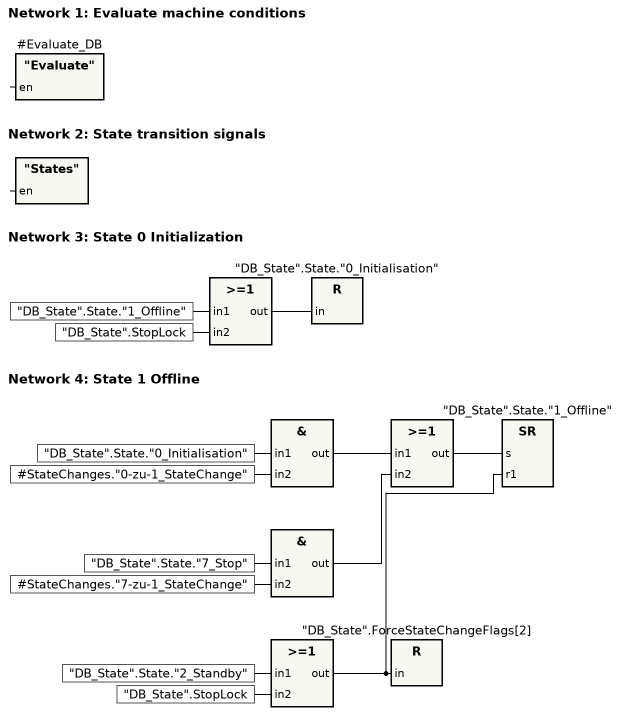
   #Evaluate_DB();   // "Evaluate"
END_REGION

REGION Network 2: State transition signals
   "States"();
END_REGION

REGION Network 3: State 0 Initialization
   // The "missing" SET logic is here:
   // Initialise (FB25) NW 2: "DB_StateMachine".State."0_Initialisation" := TRUE;
   IF "DB_State".State."1_Offline" OR "DB_State".StopLock THEN
       "DB_State".State."0_Initialisation" := FALSE;
   END_IF;
END_REGION

REGION Network 4: State 1 Offline
   #_w1 := "DB_State".State."2_Standby" OR "DB_State".StopLock;
   IF ("DB_State".State."0_Initialisation" AND #StateChanges."0-zu-1_StateChange") OR ("DB_State".State."7_Stop" AND #StateChanges."7-zu-1_StateChange") THEN
       "DB_State".State."1_Offline" := TRUE;   // SR flip-flop
   END_IF;
   IF #_w1 THEN
       "DB_State".State."1_Offline" := FALSE;
       "DB_State".ForceStateChangeFlags[2] := FALSE;
   END_IF;
END_REGION

REGION Network 5: State 2 Standby
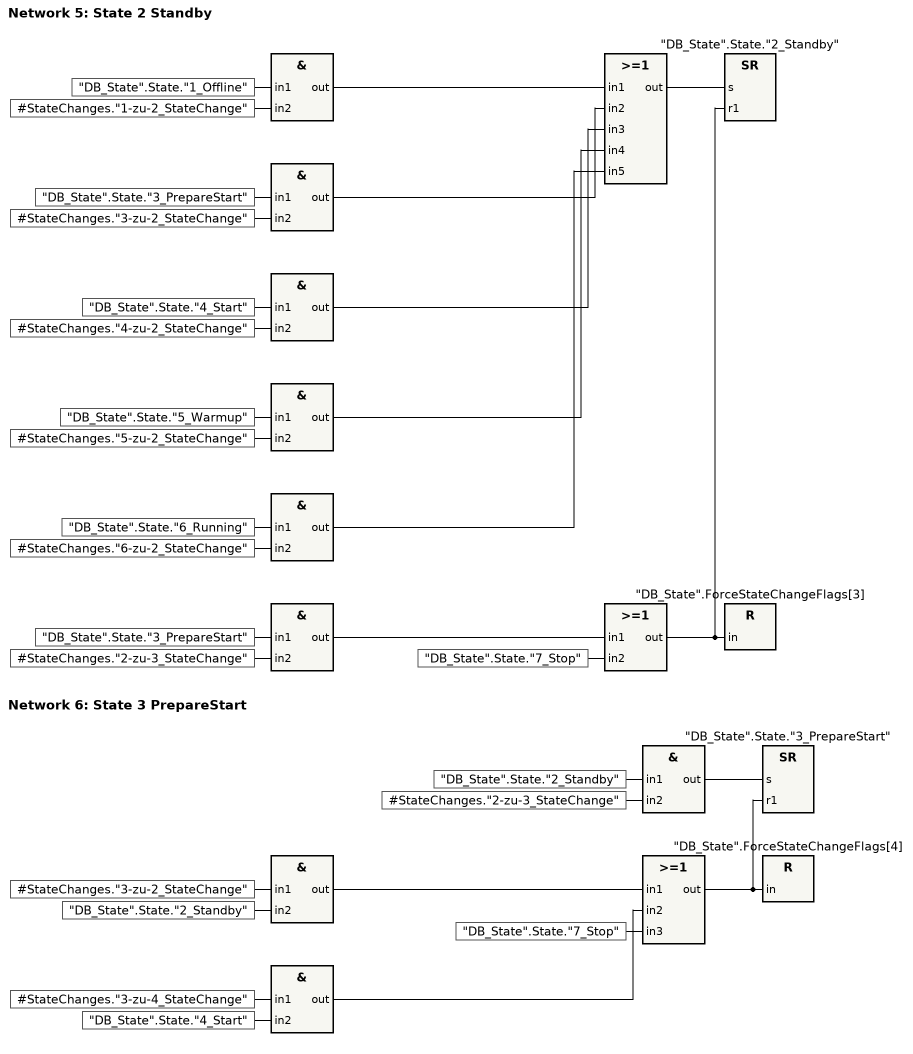
   #_w1 := ("DB_State".State."3_PrepareStart" AND #StateChanges."2-zu-3_StateChange") OR "DB_State".State."7_Stop";
   IF ("DB_State".State."1_Offline" AND #StateChanges."1-zu-2_StateChange") OR ("DB_State".State."3_PrepareStart" AND #StateChanges."3-zu-2_StateChange") OR ("DB_State".State."4_Start" AND #StateChanges."4-zu-2_StateChange") OR ("DB_State".State."5_Warmup" AND #StateChanges."5-zu-2_StateChange") OR ("DB_State".State."6_Running" AND #StateChanges."6-zu-2_StateChange") THEN
       "DB_State".State."2_Standby" := TRUE;   // SR flip-flop
   END_IF;
   IF #_w1 THEN
       "DB_State".State."2_Standby" := FALSE;
       "DB_State".ForceStateChangeFlags[3] := FALSE;
   END_IF;
END_REGION

REGION Network 6: State 3 PrepareStart
   #_w1 := (#StateChanges."3-zu-2_StateChange" AND "DB_State".State."2_Standby") OR (#StateChanges."3-zu-4_StateChange" AND "DB_State".State."4_Start") OR "DB_State".State."7_Stop";
   IF "DB_State".State."2_Standby" AND #StateChanges."2-zu-3_StateChange" THEN
       "DB_State".State."3_PrepareStart" := TRUE;   // SR flip-flop
   END_IF;
   IF #_w1 THEN
       "DB_State".State."3_PrepareStart" := FALSE;
       "DB_State".ForceStateChangeFlags[4] := FALSE;
   END_IF;
END_REGION

REGION Network 7: State 4 Start
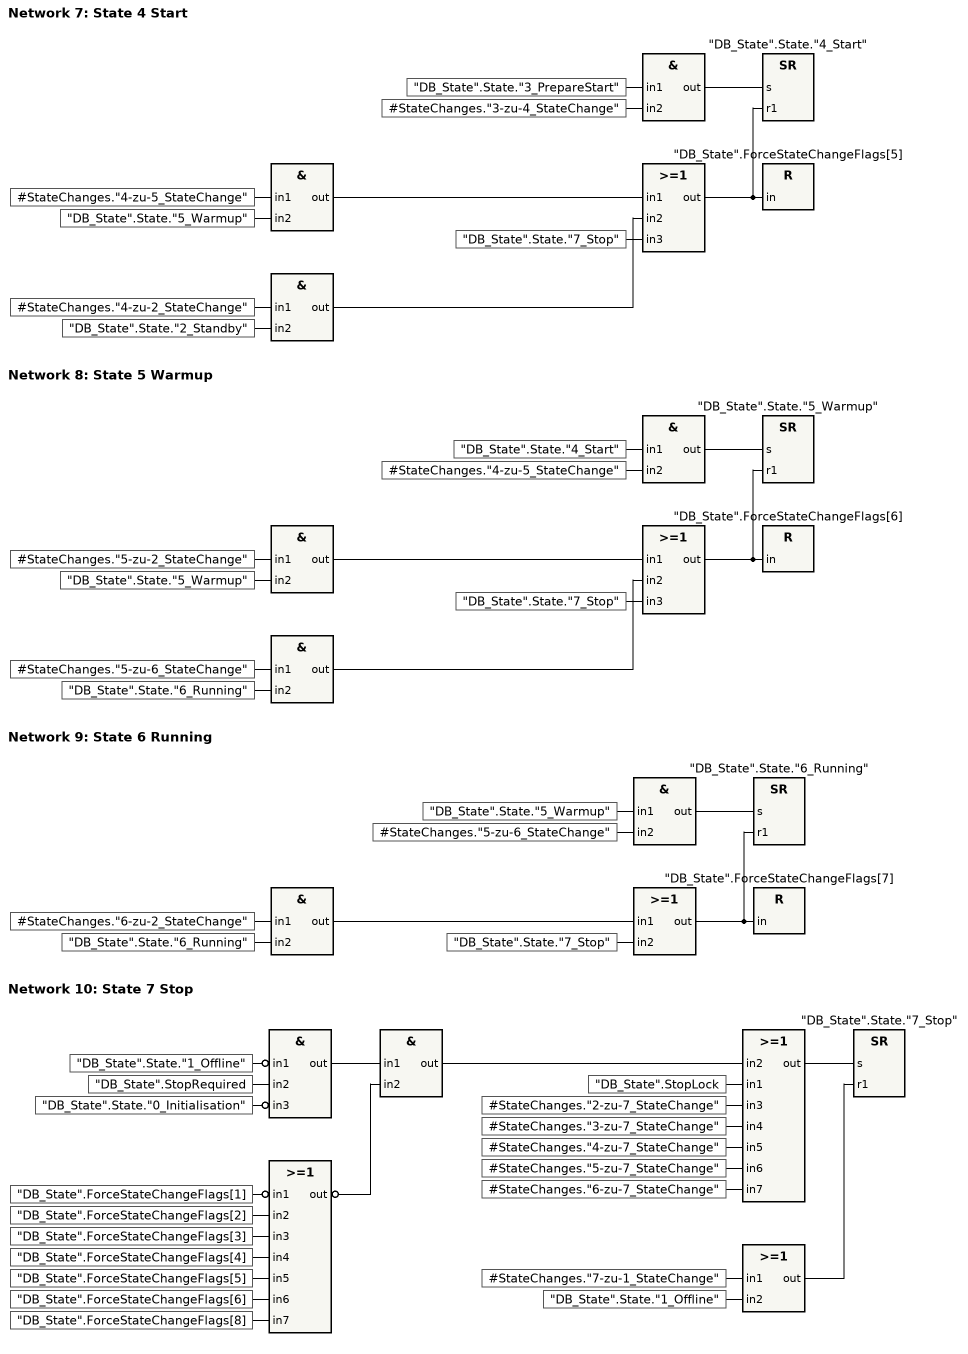
   #_w1 := (#StateChanges."4-zu-5_StateChange" AND "DB_State".State."5_Warmup") OR (#StateChanges."4-zu-2_StateChange" AND "DB_State".State."2_Standby") OR "DB_State".State."7_Stop";
   IF "DB_State".State."3_PrepareStart" AND #StateChanges."3-zu-4_StateChange" THEN
       "DB_State".State."4_Start" := TRUE;   // SR flip-flop
   END_IF;
   IF #_w1 THEN
       "DB_State".State."4_Start" := FALSE;
       "DB_State".ForceStateChangeFlags[5] := FALSE;
   END_IF;
END_REGION

REGION Network 8: State 5 Warmup
   #_w1 := (#StateChanges."5-zu-2_StateChange" AND "DB_State".State."5_Warmup") OR (#StateChanges."5-zu-6_StateChange" AND "DB_State".State."6_Running") OR "DB_State".State."7_Stop";
   IF "DB_State".State."4_Start" AND #StateChanges."4-zu-5_StateChange" THEN
       "DB_State".State."5_Warmup" := TRUE;   // SR flip-flop
   END_IF;
   IF #_w1 THEN
       "DB_State".State."5_Warmup" := FALSE;
       "DB_State".ForceStateChangeFlags[6] := FALSE;
   END_IF;
END_REGION

REGION Network 9: State 6 Running
   #_w1 := (#StateChanges."6-zu-2_StateChange" AND "DB_State".State."6_Running") OR "DB_State".State."7_Stop";
   IF "DB_State".State."5_Warmup" AND #StateChanges."5-zu-6_StateChange" THEN
       "DB_State".State."6_Running" := TRUE;   // SR flip-flop
   END_IF;
   IF #_w1 THEN
       "DB_State".State."6_Running" := FALSE;
       "DB_State".ForceStateChangeFlags[7] := FALSE;
   END_IF;
END_REGION

REGION Network 10: State 7 Stop
   IF (NOT "DB_State".State."1_Offline" AND "DB_State".StopRequired AND NOT "DB_State".State."0_Initialisation" AND NOT (NOT "DB_State".ForceStateChangeFlags[1] OR "DB_State".ForceStateChangeFlags[2] OR "DB_State".ForceStateChangeFlags[3] OR "DB_State".ForceStateChangeFlags[4] OR "DB_State".ForceStateChangeFlags[5] OR "DB_State".ForceStateChangeFlags[6] OR "DB_State".ForceStateChangeFlags[8])) OR "DB_State".StopLock OR #StateChanges."2-zu-7_StateChange" OR #StateChanges."3-zu-7_StateChange" OR #StateChanges."4-zu-7_StateChange" OR #StateChanges."5-zu-7_StateChange" OR #StateChanges."6-zu-7_StateChange" THEN
       "DB_State".State."7_Stop" := TRUE;   // SR flip-flop
   END_IF;
   IF #StateChanges."7-zu-1_StateChange" OR "DB_State".State."1_Offline" THEN
       "DB_State".State."7_Stop" := FALSE;
   END_IF;
END_REGION
END_FUNCTION_BLOCK

FUNCTION_BLOCK "Evaluate"   // FB26, FBD
TITLE = Evaluate machine state conditions
{ S7_Optimized_Access := 'TRUE' }
AUTHOR : Heaten
VERSION : 0.1
// stored: AutoNumber true, IsIECCheckEnabled false, IsRetainMemResEnabled false, MemoryReserve 0, SetENOAutomatically false, UDAEnableTagReadback false
   VAR
      TOF2_StandbyPauseTime { S7_SetPoint := 'True'} : TOF_TIME;
      TON2_Standby { S7_SetPoint := 'True'} : TON_TIME;
      TON3_PrepareStart { S7_SetPoint := 'True'} : TON_TIME;
      TON4_Start { S7_SetPoint := 'True'} : TON_TIME;
      TON5_Warmup { S7_SetPoint := 'True'} : TON_TIME;
      TON7_Stop { S7_SetPoint := 'True'} : TON_TIME;
      MinimumPriming { S7_SetPoint := 'True'} : TON_TIME;
   END_VAR
   VAR_TEMP
      HydrolockSpeed : Real;
      HeatSinkTemperatureMax : Real;
   END_VAR
BEGIN

REGION Network 1: Check running condition: system initialized
   // Add more conditions here
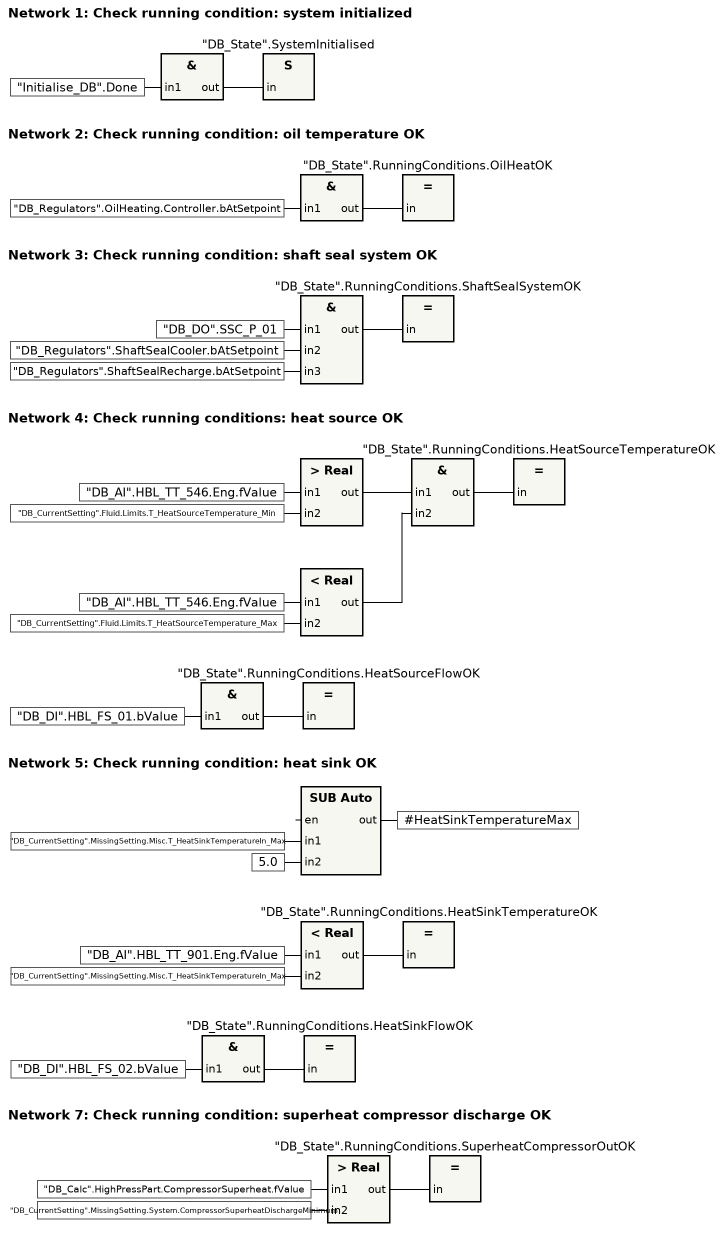
   IF "Initialise_DB".Done THEN "DB_State".SystemInitialised := TRUE; END_IF;
END_REGION

REGION Network 2: Check running condition: oil temperature OK
   "DB_State".RunningConditions.OilHeatOK := "DB_Regulators".OilHeating.Controller.bAtSetpoint;
END_REGION

REGION Network 3: Check running condition: shaft seal system OK
   "DB_State".RunningConditions.ShaftSealSystemOK := "DB_DO".SSC_P_01 AND "DB_Regulators".ShaftSealCooler.bAtSetpoint AND "DB_Regulators".ShaftSealRecharge.bAtSetpoint;
END_REGION

REGION Network 4: Check running conditions: heat source OK
   "DB_State".RunningConditions.HeatSourceTemperatureOK := ("DB_AI".HBL_TT_546.Eng.fValue > "DB_CurrentSetting".Fluid.Limits.T_HeatSourceTemperature_Min) AND ("DB_AI".HBL_TT_546.Eng.fValue < "DB_CurrentSetting".Fluid.Limits.T_HeatSourceTemperature_Max);
   "DB_State".RunningConditions.HeatSourceFlowOK := "DB_DI".HBL_FS_01.bValue;
END_REGION

REGION Network 5: Check running condition: heat sink OK
   // NOTE: leave a little headroom to the limit for standby, otherwise the machine shuts down (via alarm 2101) at the same temperature as it should go to standby on
   #HeatSinkTemperatureMax := "DB_CurrentSetting".MissingSetting.Misc.T_HeatSinkTemperatureIn_Max - 5.0;
   "DB_State".RunningConditions.HeatSinkTemperatureOK := "DB_AI".HBL_TT_901.Eng.fValue < "DB_CurrentSetting".MissingSetting.Misc.T_HeatSinkTemperatureIn_Max;
   "DB_State".RunningConditions.HeatSinkFlowOK := "DB_DI".HBL_FS_02.bValue;
END_REGION

REGION Network 6 (SCL): Check running condition: recuperator working
   // Recuperator sits between evaporator and compressor and SHOULD INCREASE THE SUPERHEAT (ie delta T over the recuperator should be positive)
   // 
   // Recuperator window: must add at least "DB_CurrentSetting".MissingSetting.System.RecuperatorSuperheatGainWorking degrees to be considered working, 
   // but can then fall as low as "DB_CurrentSetting".MissingSetting.System.RecuperatorSuperheatGainNotWorking degrees before it is considered not working again
   (*
   IF ("DB_Calc".LowPressPart.CompressorSuperheat.fValue - 2) <      //If the superheat at compressor inlet minus 2 is smaller than
       "DB_Calc".LowPressPart.EvaporatorSuperheat.fValue THEN          //the superheat at the evaporator, the recuperator doesn´t work
       "StateMachine_DB".RunningConditions.RecuperatorWorking := FALSE;
   ELSIF
       ("DB_Calc".LowPressPart.CompressorSuperheat.fValue + 3) >     //If the superheat at compressor inlet plus 3 is bigger than
       "DB_Calc".LowPressPart.EvaporatorSuperheat.fValue THEN          //the superheat at the evaporator, the recuperator works
       "StateMachine_DB".RunningConditions.RecuperatorWorking := TRUE;
   END_IF;
   *)

   // Rewritten with user-defined limits and right-side-up logic
   // Also don't evaluate the condition unless it's relevant, to avoid odd conditions during earlier states/cold start setting this accidentally
   IF "DB_State".State.State_Number = 5 OR "DB_State".State.State_Number = 6 THEN
       IF "DB_Calc".LowPressPart.CompressorSuperheat.fValue > "DB_Calc".LowPressPart.EvaporatorSuperheat.fValue + "DB_CurrentSetting".MissingSetting.System.RecuperatorDeltaTWorking THEN
           "DB_State".RunningConditions.RecuperatorWorking := TRUE;
       ELSIF "DB_Calc".LowPressPart.CompressorSuperheat.fValue < "DB_Calc".LowPressPart.EvaporatorSuperheat.fValue + "DB_CurrentSetting".MissingSetting.System.RecuperatorDeltaTNotWorking THEN
           "DB_State".RunningConditions.RecuperatorWorking := FALSE;
       END_IF;
   ELSE
       "DB_State".RunningConditions.RecuperatorWorking := FALSE;
   END_IF;
END_REGION

REGION Network 7: Check running condition: superheat compressor discharge OK
   "DB_State".RunningConditions.SuperheatCompressorOutOK := "DB_Calc".HighPressPart.CompressorSuperheat.fValue > "DB_CurrentSetting".MissingSetting.System.CompressorSuperheatDischargeMinimum;
END_REGION

REGION Network 8: Check running condition: at or above hydrolock speed
   // Give a small margin for error, so if it sits at, for example 288.2 RPM and the limit is 290, it will work.
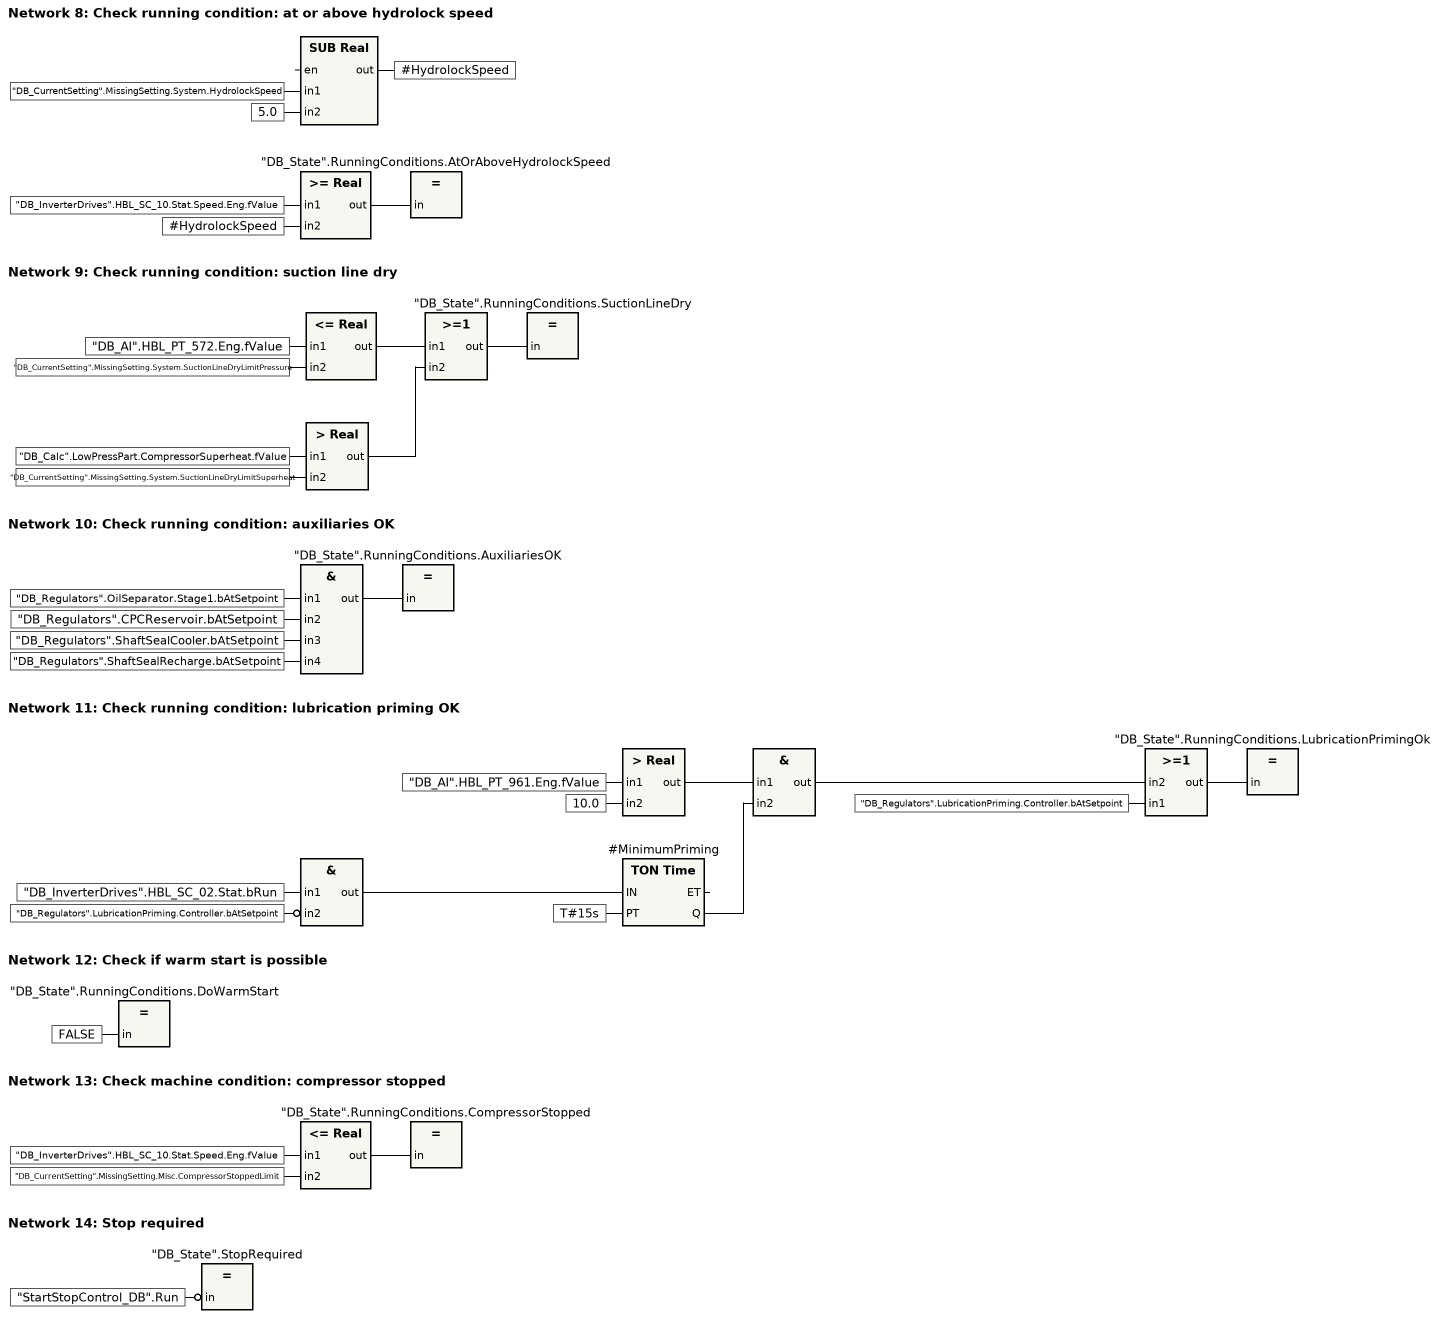
   #HydrolockSpeed := "DB_CurrentSetting".MissingSetting.System.HydrolockSpeed - 5.0;
   "DB_State".RunningConditions.AtOrAboveHydrolockSpeed := "DB_InverterDrives".HBL_SC_10.Stat.Speed.Eng.fValue >= #HydrolockSpeed;
END_REGION

REGION Network 9: Check running condition: suction line dry
   "DB_State".RunningConditions.SuctionLineDry := ("DB_AI".HBL_PT_572.Eng.fValue <= "DB_CurrentSetting".MissingSetting.System.SuctionLineDryLimitPressure) OR ("DB_Calc".LowPressPart.CompressorSuperheat.fValue > "DB_CurrentSetting".MissingSetting.System.SuctionLineDryLimitSuperheat);
END_REGION

REGION Network 10: Check running condition: auxiliaries OK
   "DB_State".RunningConditions.AuxiliariesOK := "DB_Regulators".OilSeparator.Stage1.bAtSetpoint AND "DB_Regulators".CPCReservoir.bAtSetpoint AND "DB_Regulators".ShaftSealCooler.bAtSetpoint AND "DB_Regulators".ShaftSealRecharge.bAtSetpoint;
END_REGION

REGION Network 11: Check running condition: lubrication priming OK
   // The simplest is to just look at the regulator's .bAtSetpoint bit. But the lubrication priming pump may be too small to reach the setpoint. So a hybrid condition is:
   // IF the pressure is at setpoint OR
   // the motor has been running for at least X sec when not at setpoint AND 
   // the developed lubrication pressure is greater than Y kPa THEN
   // the lubrication system is working ok.
   // NOTE: hardcoded params = bad!!
   #MinimumPriming(IN := "DB_InverterDrives".HBL_SC_02.Stat.bRun AND NOT "DB_Regulators".LubricationPriming.Controller.bAtSetpoint,   // TON
                   PT := T#15s);
   "DB_State".RunningConditions.LubricationPrimingOk := (("DB_AI".HBL_PT_961.Eng.fValue > 10.0) AND #MinimumPriming.Q) OR "DB_Regulators".LubricationPriming.Controller.bAtSetpoint;
END_REGION

REGION Network 12: Check if warm start is possible
   // Think of an appropriate condition
   "DB_State".RunningConditions.DoWarmStart := FALSE;
END_REGION

REGION Network 13: Check machine condition: compressor stopped
   "DB_State".RunningConditions.CompressorStopped := "DB_InverterDrives".HBL_SC_10.Stat.Speed.Eng.fValue <= "DB_CurrentSetting".MissingSetting.Misc.CompressorStoppedLimit;
END_REGION

REGION Network 14: Stop required
   // NOte: stop conditions are evaluated by FB30 StartStopControl
   "DB_State".StopRequired := NOT "StartStopControl_DB".Run;
END_REGION

REGION Network 15: Check for risk of hydrolock
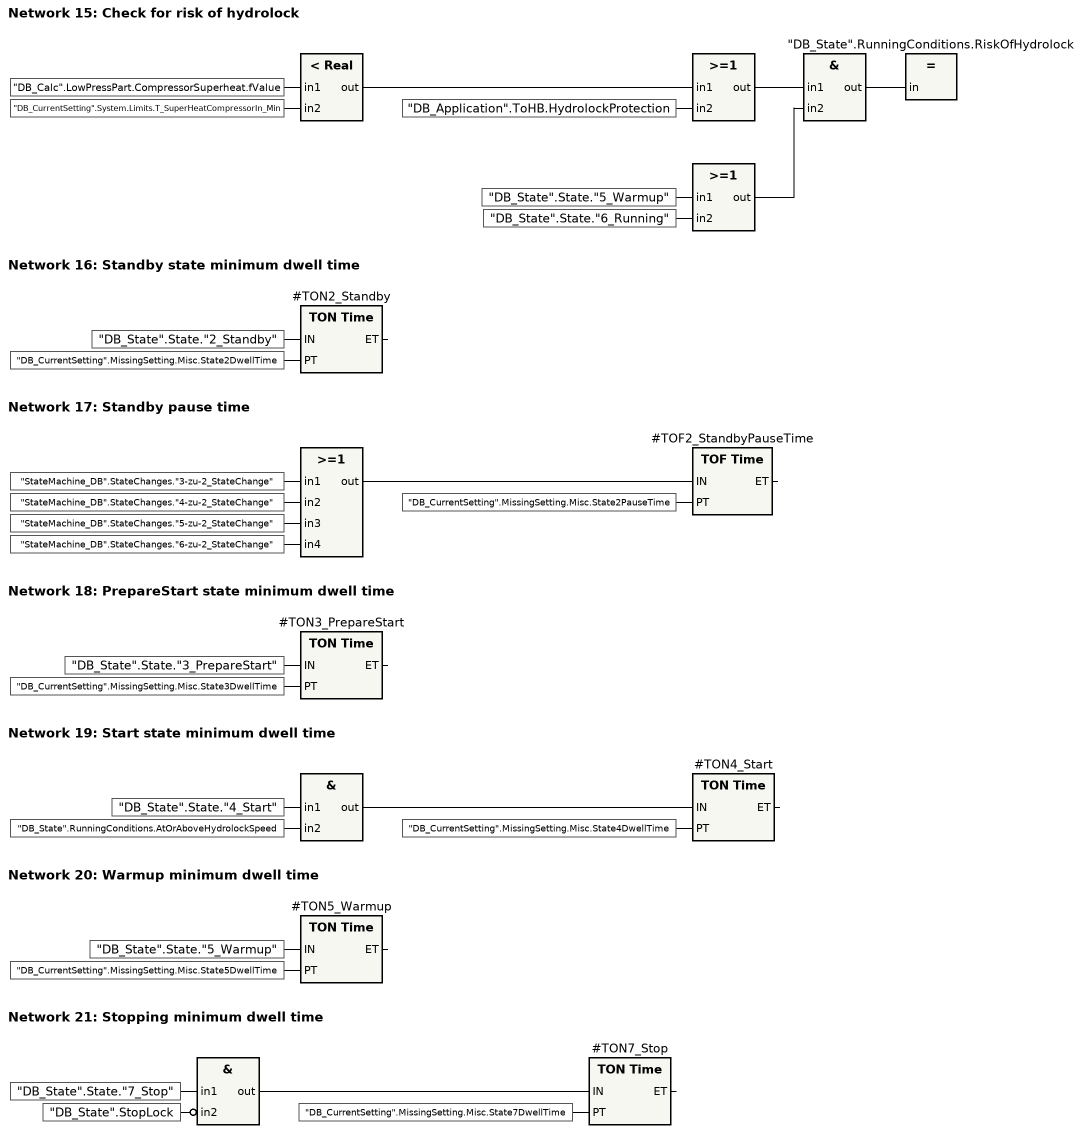
   "DB_State".RunningConditions.RiskOfHydrolock := (("DB_Calc".LowPressPart.CompressorSuperheat.fValue < "DB_CurrentSetting".System.Limits.T_SuperHeatCompressorIn_Min) OR "DB_Application".ToHB.HydrolockProtection) AND ("DB_State".State."5_Warmup" OR "DB_State".State."6_Running");
END_REGION

REGION Network 16: Standby state minimum dwell time
   #TON2_Standby(IN := "DB_State".State."2_Standby",   // TON
                 PT := "DB_CurrentSetting".MissingSetting.Misc.State2DwellTime);
END_REGION

REGION Network 17: Standby pause time
   // Minimum pause in Standby before resume
   #TOF2_StandbyPauseTime(IN := "StateMachine_DB".StateChanges."3-zu-2_StateChange" OR "StateMachine_DB".StateChanges."4-zu-2_StateChange" OR "StateMachine_DB".StateChanges."5-zu-2_StateChange" OR "StateMachine_DB".StateChanges."6-zu-2_StateChange",   // TOF
                          PT := "DB_CurrentSetting".MissingSetting.Misc.State2PauseTime);
END_REGION

REGION Network 18: PrepareStart state minimum dwell time
   #TON3_PrepareStart(IN := "DB_State".State."3_PrepareStart",   // TON
                      PT := "DB_CurrentSetting".MissingSetting.Misc.State3DwellTime);
END_REGION

REGION Network 19: Start state minimum dwell time
   #TON4_Start(IN := "DB_State".State."4_Start" AND "DB_State".RunningConditions.AtOrAboveHydrolockSpeed,   // TON
               PT := "DB_CurrentSetting".MissingSetting.Misc.State4DwellTime);
END_REGION

REGION Network 20: Warmup minimum dwell time
   #TON5_Warmup(IN := "DB_State".State."5_Warmup",   // TON
                PT := "DB_CurrentSetting".MissingSetting.Misc.State5DwellTime);
END_REGION

REGION Network 21: Stopping minimum dwell time
   #TON7_Stop(IN := "DB_State".State."7_Stop" AND NOT "DB_State".StopLock,   // TON
              PT := "DB_CurrentSetting".MissingSetting.Misc.State7DwellTime);
END_REGION
END_FUNCTION_BLOCK

FUNCTION "States" : Void   // FC27, FBD
TITLE = State change signal generation
{ S7_Optimized_Access := 'TRUE' }
VERSION : 0.1
// stored: AutoNumber true, IsIECCheckEnabled false, SetENOAutomatically false, UDAEnableTagReadback false
BEGIN

REGION Network 1: State 0 Initialization
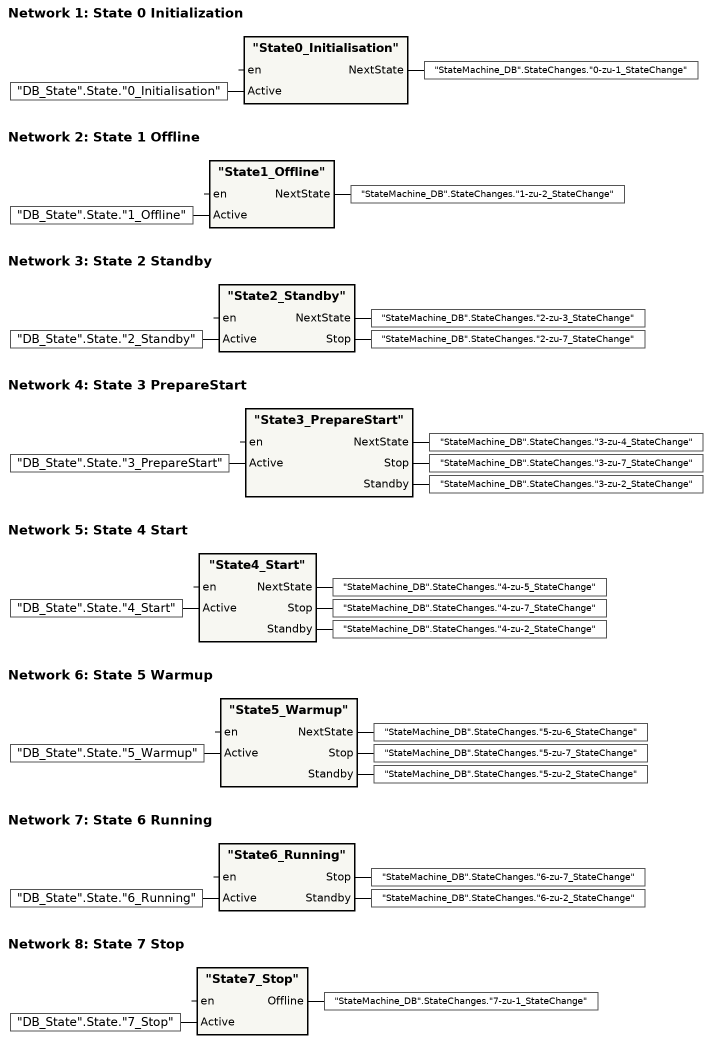
   "State0_Initialisation"(Active := "DB_State".State."0_Initialisation",
                           NextState => "StateMachine_DB".StateChanges."0-zu-1_StateChange");
END_REGION

REGION Network 2: State 1 Offline
   "State1_Offline"(Active := "DB_State".State."1_Offline",
                    NextState => "StateMachine_DB".StateChanges."1-zu-2_StateChange");
END_REGION

REGION Network 3: State 2 Standby
   "State2_Standby"(Active := "DB_State".State."2_Standby",
                    NextState => "StateMachine_DB".StateChanges."2-zu-3_StateChange",
                    Stop => "StateMachine_DB".StateChanges."2-zu-7_StateChange");
END_REGION

REGION Network 4: State 3 PrepareStart
   "State3_PrepareStart"(Active := "DB_State".State."3_PrepareStart",
                         NextState => "StateMachine_DB".StateChanges."3-zu-4_StateChange",
                         Stop => "StateMachine_DB".StateChanges."3-zu-7_StateChange",
                         Standby => "StateMachine_DB".StateChanges."3-zu-2_StateChange");
END_REGION

REGION Network 5: State 4 Start
   "State4_Start"(Active := "DB_State".State."4_Start",
                  NextState => "StateMachine_DB".StateChanges."4-zu-5_StateChange",
                  Stop => "StateMachine_DB".StateChanges."4-zu-7_StateChange",
                  Standby => "StateMachine_DB".StateChanges."4-zu-2_StateChange");
END_REGION

REGION Network 6: State 5 Warmup
   "State5_Warmup"(Active := "DB_State".State."5_Warmup",
                   NextState => "StateMachine_DB".StateChanges."5-zu-6_StateChange",
                   Stop => "StateMachine_DB".StateChanges."5-zu-7_StateChange",
                   Standby => "StateMachine_DB".StateChanges."5-zu-2_StateChange");
END_REGION

REGION Network 7: State 6 Running
   "State6_Running"(Active := "DB_State".State."6_Running",
                    Stop => "StateMachine_DB".StateChanges."6-zu-7_StateChange",
                    Standby => "StateMachine_DB".StateChanges."6-zu-2_StateChange");
END_REGION

REGION Network 8: State 7 Stop
   "State7_Stop"(Active := "DB_State".State."7_Stop",
                 Offline => "StateMachine_DB".StateChanges."7-zu-1_StateChange");
END_REGION
END_FUNCTION

FUNCTION "State0_Initialisation" : Void   // FC1, FBD
{ S7_Optimized_Access := 'TRUE' }
VERSION : 0.1
// stored: AutoNumber true, IsIECCheckEnabled false, SetENOAutomatically false, UDAEnableTagReadback false
   VAR_INPUT
      Active : Bool;
   END_VAR
   VAR_OUTPUT
      NextState : Bool;
   END_VAR
BEGIN

REGION Network 1: State number
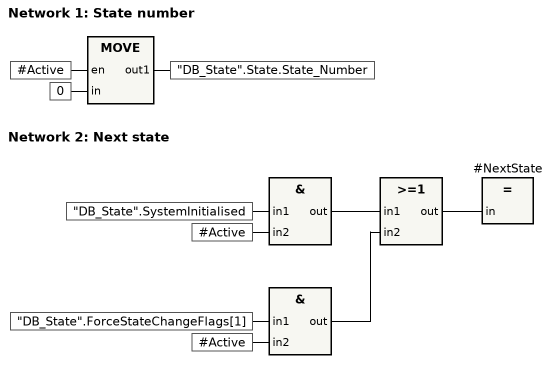
   IF #Active THEN "DB_State".State.State_Number := 0; END_IF;
END_REGION

REGION Network 2: Next state
   #NextState := ("DB_State".SystemInitialised AND #Active) OR ("DB_State".ForceStateChangeFlags[1] AND #Active);
END_REGION
END_FUNCTION

FUNCTION "State1_Offline" : Void   // FC4, FBD
{ S7_Optimized_Access := 'TRUE' }
VERSION : 0.1
// stored: AutoNumber true, IsIECCheckEnabled false, SetENOAutomatically false, UDAEnableTagReadback false
   VAR_INPUT
      Active : Bool;
   END_VAR
   VAR_OUTPUT
      NextState : Bool;
   END_VAR
BEGIN

REGION Network 1: State number
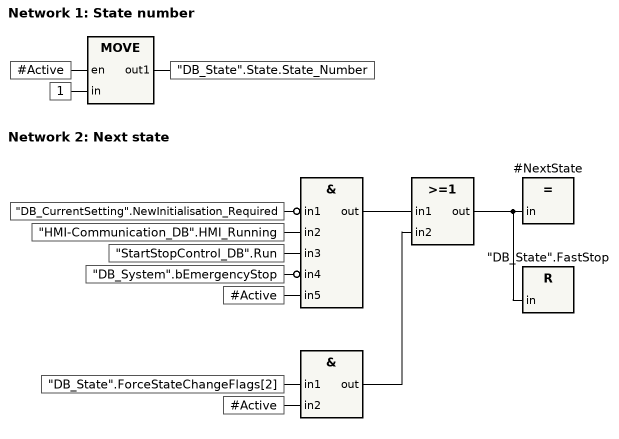
   IF #Active THEN "DB_State".State.State_Number := 1; END_IF;
END_REGION

REGION Network 2: Next state
   #NextState := (NOT "DB_CurrentSetting".NewInitialisation_Required AND "HMI-Communication_DB".HMI_Running AND "StartStopControl_DB".Run AND NOT "DB_System".bEmergencyStop AND #Active) OR ("DB_State".ForceStateChangeFlags[2] AND #Active);
   IF #NextState THEN "DB_State".FastStop := FALSE; END_IF;
END_REGION
END_FUNCTION

FUNCTION "State2_Standby" : Void   // FC9, FBD
{ S7_Optimized_Access := 'TRUE' }
VERSION : 0.1
// stored: AutoNumber true, IsIECCheckEnabled false, SetENOAutomatically false, UDAEnableTagReadback false
   VAR_INPUT
      Active : Bool;
   END_VAR
   VAR_OUTPUT
      NextState : Bool;
      Stop : Bool;
   END_VAR
   VAR_TEMP
      NextStateConditions : Bool;
      PauseHere : Bool;
   END_VAR
   VAR_TEMP   // added for the SCL form of the ladder/FBD networks
      _w1 : Bool;
   END_VAR
BEGIN

REGION Network 1: State number
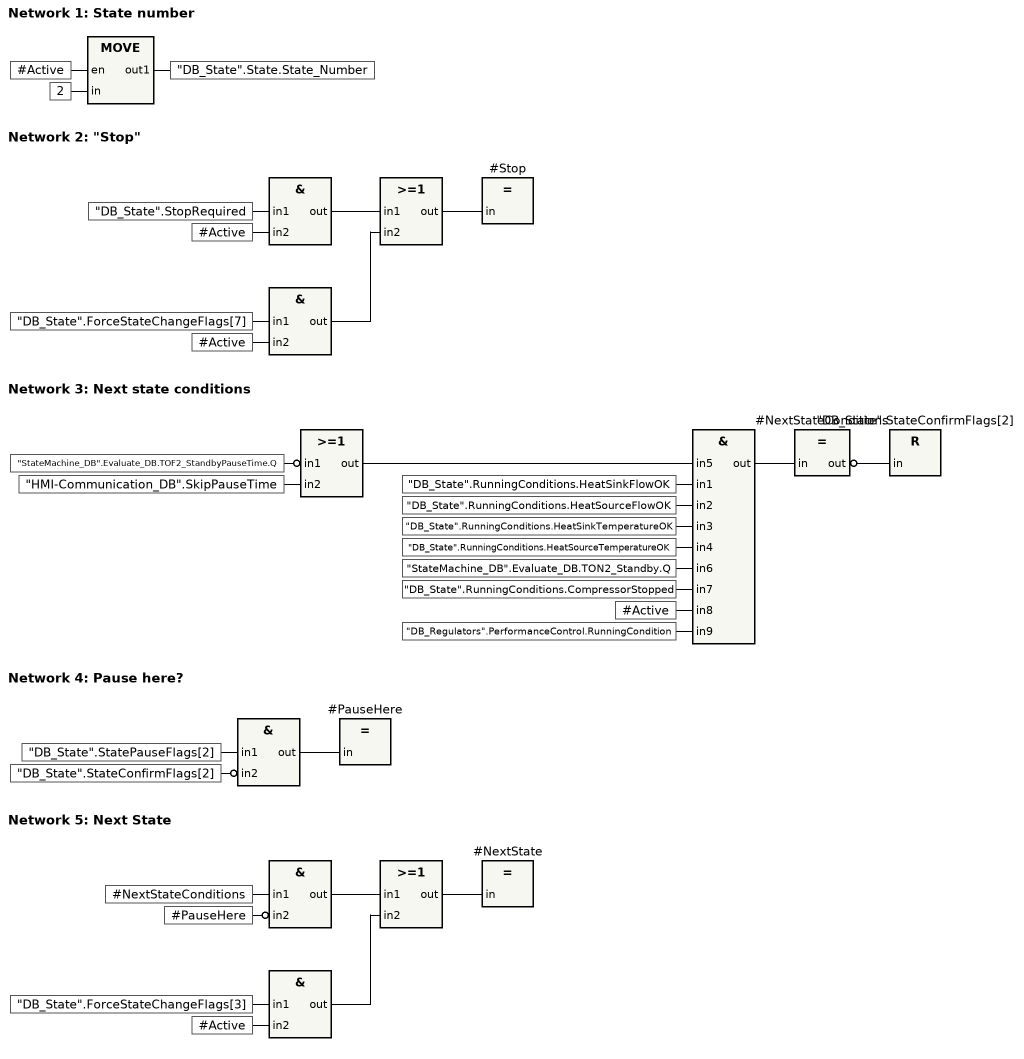
   IF #Active THEN "DB_State".State.State_Number := 2; END_IF;
END_REGION

REGION Network 2: "Stop"
   #Stop := ("DB_State".StopRequired AND #Active) OR ("DB_State".ForceStateChangeFlags[7] AND #Active);
END_REGION

REGION Network 3: Next state conditions
   #_w1 := (NOT "StateMachine_DB".Evaluate_DB.TOF2_StandbyPauseTime.Q OR "HMI-Communication_DB".SkipPauseTime) AND "DB_State".RunningConditions.HeatSinkFlowOK AND "DB_State".RunningConditions.HeatSourceFlowOK AND "DB_State".RunningConditions.HeatSinkTemperatureOK AND "DB_State".RunningConditions.HeatSourceTemperatureOK AND "StateMachine_DB".Evaluate_DB.TON2_Standby.Q AND "DB_State".RunningConditions.CompressorStopped AND #Active AND "DB_Regulators".PerformanceControl.RunningCondition;
   #NextStateConditions := #_w1;
   IF NOT #_w1 THEN "DB_State".StateConfirmFlags[2] := FALSE; END_IF;
END_REGION

REGION Network 4: Pause here?
   // Pause   Confirm  PauseHere
   // 0            0              0
   // 0            1              0
   // 1            0              1
   // 1            1              0
   #PauseHere := "DB_State".StatePauseFlags[2] AND NOT "DB_State".StateConfirmFlags[2];
END_REGION

REGION Network 5: Next State
   #NextState := (#NextStateConditions AND NOT #PauseHere) OR ("DB_State".ForceStateChangeFlags[3] AND #Active);
END_REGION
END_FUNCTION

FUNCTION "State3_PrepareStart" : Void   // FC36, FBD
{ S7_Optimized_Access := 'TRUE' }
VERSION : 0.1
// stored: AutoNumber true, IsIECCheckEnabled false, SetENOAutomatically false, UDAEnableTagReadback false
   VAR_INPUT
      Active : Bool;
   END_VAR
   VAR_OUTPUT
      NextState : Bool;
      Stop : Bool;
      Standby : Bool;
   END_VAR
   VAR_TEMP
      NextStateConditions : Bool;
      PauseHere : Bool;
   END_VAR
   VAR_TEMP   // added for the SCL form of the ladder/FBD networks
      _w1 : Bool;
   END_VAR
BEGIN

REGION Network 1: State number
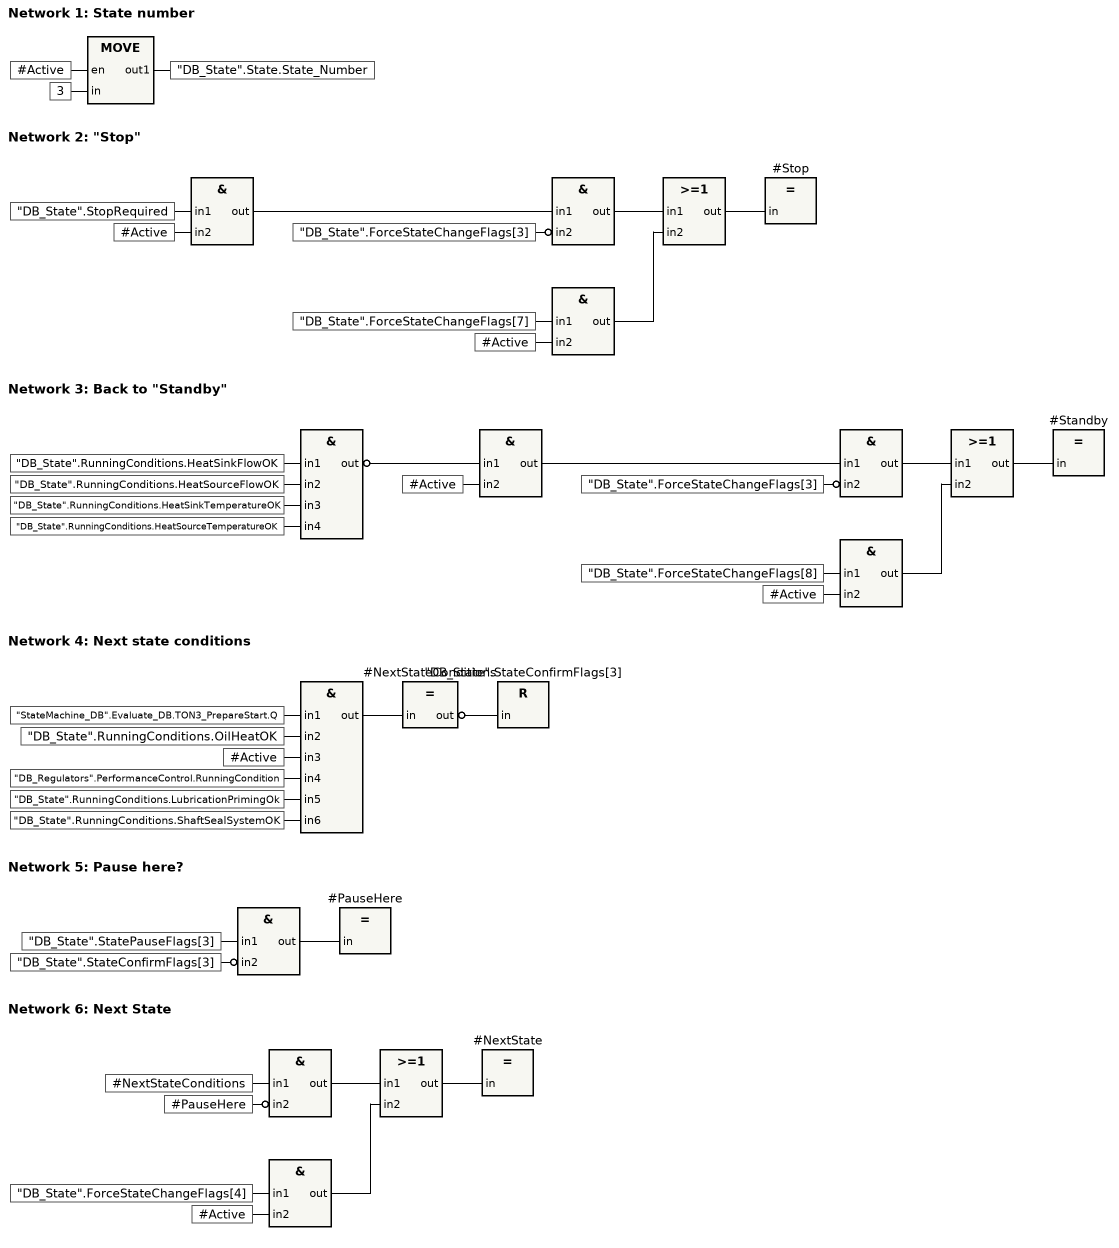
   IF #Active THEN "DB_State".State.State_Number := 3; END_IF;
END_REGION

REGION Network 2: "Stop"
   #Stop := ("DB_State".StopRequired AND #Active AND NOT "DB_State".ForceStateChangeFlags[3]) OR ("DB_State".ForceStateChangeFlags[7] AND #Active);
END_REGION

REGION Network 3: Back to "Standby"
   #Standby := (NOT ("DB_State".RunningConditions.HeatSinkFlowOK AND "DB_State".RunningConditions.HeatSourceFlowOK AND "DB_State".RunningConditions.HeatSinkTemperatureOK AND "DB_State".RunningConditions.HeatSourceTemperatureOK) AND #Active AND NOT "DB_State".ForceStateChangeFlags[3]) OR ("DB_State".ForceStateChangeFlags[8] AND #Active);
END_REGION

REGION Network 4: Next state conditions
   #_w1 := "StateMachine_DB".Evaluate_DB.TON3_PrepareStart.Q AND "DB_State".RunningConditions.OilHeatOK AND #Active AND "DB_Regulators".PerformanceControl.RunningCondition AND "DB_State".RunningConditions.LubricationPrimingOk AND "DB_State".RunningConditions.ShaftSealSystemOK;
   #NextStateConditions := #_w1;
   IF NOT #_w1 THEN "DB_State".StateConfirmFlags[3] := FALSE; END_IF;
END_REGION

REGION Network 5: Pause here?
   // Pause   Confirm  PauseHere
   // 0            0              0
   // 0            1              0
   // 1            0              1
   // 1            1              0
   #PauseHere := "DB_State".StatePauseFlags[3] AND NOT "DB_State".StateConfirmFlags[3];
END_REGION

REGION Network 6: Next State
   #NextState := (#NextStateConditions AND NOT #PauseHere) OR ("DB_State".ForceStateChangeFlags[4] AND #Active);
END_REGION
END_FUNCTION

FUNCTION "State4_Start" : Void   // FC53, FBD
{ S7_Optimized_Access := 'TRUE' }
VERSION : 0.1
// stored: AutoNumber true, IsIECCheckEnabled false, SetENOAutomatically false, UDAEnableTagReadback false
   VAR_INPUT
      Active : Bool;
   END_VAR
   VAR_OUTPUT
      NextState : Bool;
      Stop : Bool;
      Standby : Bool;
   END_VAR
   VAR_TEMP
      NextStateConditions : Bool;
      PauseHere : Bool;
   END_VAR
   VAR_TEMP   // added for the SCL form of the ladder/FBD networks
      _w1 : Bool;
   END_VAR
BEGIN

REGION Network 1: State number
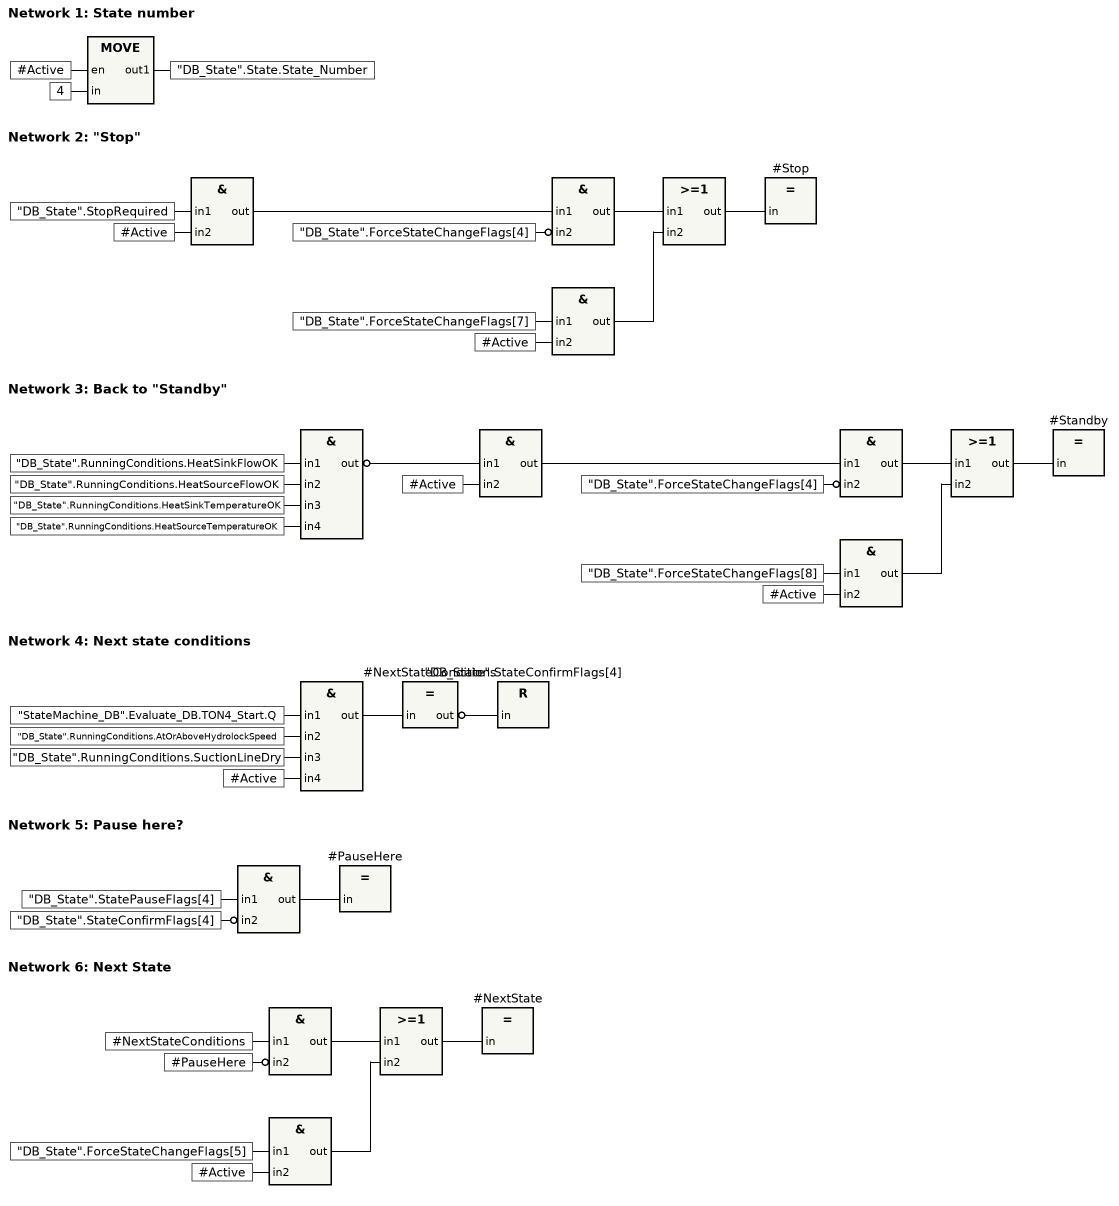
   IF #Active THEN "DB_State".State.State_Number := 4; END_IF;
END_REGION

REGION Network 2: "Stop"
   #Stop := ("DB_State".StopRequired AND #Active AND NOT "DB_State".ForceStateChangeFlags[4]) OR ("DB_State".ForceStateChangeFlags[7] AND #Active);
END_REGION

REGION Network 3: Back to "Standby"
   #Standby := (NOT ("DB_State".RunningConditions.HeatSinkFlowOK AND "DB_State".RunningConditions.HeatSourceFlowOK AND "DB_State".RunningConditions.HeatSinkTemperatureOK AND "DB_State".RunningConditions.HeatSourceTemperatureOK) AND #Active AND NOT "DB_State".ForceStateChangeFlags[4]) OR ("DB_State".ForceStateChangeFlags[8] AND #Active);
END_REGION

REGION Network 4: Next state conditions
   #_w1 := "StateMachine_DB".Evaluate_DB.TON4_Start.Q AND "DB_State".RunningConditions.AtOrAboveHydrolockSpeed AND "DB_State".RunningConditions.SuctionLineDry AND #Active;
   #NextStateConditions := #_w1;
   IF NOT #_w1 THEN "DB_State".StateConfirmFlags[4] := FALSE; END_IF;
END_REGION

REGION Network 5: Pause here?
   // Pause   Confirm  PauseHere
   // 0            0              0
   // 0            1              0
   // 1            0              1
   // 1            1              0
   #PauseHere := "DB_State".StatePauseFlags[4] AND NOT "DB_State".StateConfirmFlags[4];
END_REGION

REGION Network 6: Next State
   #NextState := (#NextStateConditions AND NOT #PauseHere) OR ("DB_State".ForceStateChangeFlags[5] AND #Active);
END_REGION
END_FUNCTION

FUNCTION "State5_Warmup" : Void   // FC55, FBD
{ S7_Optimized_Access := 'TRUE' }
VERSION : 0.1
// stored: AutoNumber true, IsIECCheckEnabled false, SetENOAutomatically false, UDAEnableTagReadback false
   VAR_INPUT
      Active : Bool;
   END_VAR
   VAR_OUTPUT
      NextState : Bool;
      Stop : Bool;
      Standby : Bool;
   END_VAR
   VAR_TEMP
      NextStateConditions : Bool;
      PauseHere : Bool;
   END_VAR
   VAR_TEMP   // added for the SCL form of the ladder/FBD networks
      _w1 : Bool;
   END_VAR
BEGIN

REGION Network 1: State number
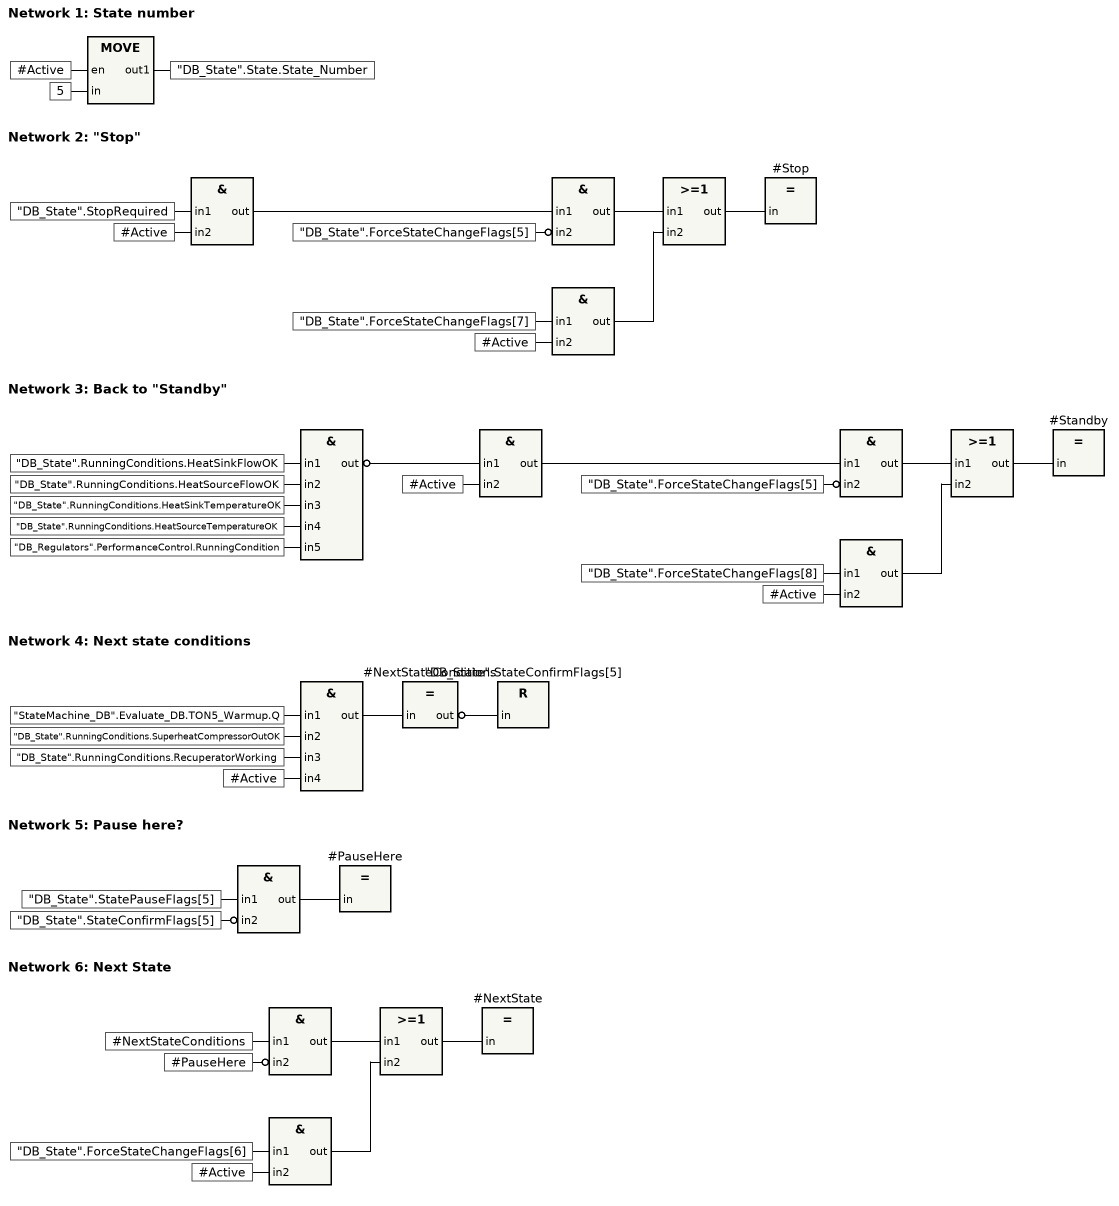
   IF #Active THEN "DB_State".State.State_Number := 5; END_IF;
END_REGION

REGION Network 2: "Stop"
   #Stop := ("DB_State".StopRequired AND #Active AND NOT "DB_State".ForceStateChangeFlags[5]) OR ("DB_State".ForceStateChangeFlags[7] AND #Active);
END_REGION

REGION Network 3: Back to "Standby"
   #Standby := (NOT ("DB_State".RunningConditions.HeatSinkFlowOK AND "DB_State".RunningConditions.HeatSourceFlowOK AND "DB_State".RunningConditions.HeatSinkTemperatureOK AND "DB_State".RunningConditions.HeatSourceTemperatureOK AND "DB_Regulators".PerformanceControl.RunningCondition) AND #Active AND NOT "DB_State".ForceStateChangeFlags[5]) OR ("DB_State".ForceStateChangeFlags[8] AND #Active);
END_REGION

REGION Network 4: Next state conditions
   #_w1 := "StateMachine_DB".Evaluate_DB.TON5_Warmup.Q AND "DB_State".RunningConditions.SuperheatCompressorOutOK AND "DB_State".RunningConditions.RecuperatorWorking AND #Active;
   #NextStateConditions := #_w1;
   IF NOT #_w1 THEN "DB_State".StateConfirmFlags[5] := FALSE; END_IF;
END_REGION

REGION Network 5: Pause here?
   // Pause   Confirm  PauseHere
   // 0            0              0
   // 0            1              0
   // 1            0              1
   // 1            1              0
   #PauseHere := "DB_State".StatePauseFlags[5] AND NOT "DB_State".StateConfirmFlags[5];
END_REGION

REGION Network 6: Next State
   #NextState := (#NextStateConditions AND NOT #PauseHere) OR ("DB_State".ForceStateChangeFlags[6] AND #Active);
END_REGION
END_FUNCTION

FUNCTION "State6_Running" : Void   // FC56, FBD
{ S7_Optimized_Access := 'TRUE' }
VERSION : 0.1
// stored: AutoNumber true, IsIECCheckEnabled false, SetENOAutomatically false, UDAEnableTagReadback false
   VAR_INPUT
      Active : Bool;
   END_VAR
   VAR_OUTPUT
      Stop : Bool;
      Standby : Bool;
   END_VAR
BEGIN

REGION Network 1: State number
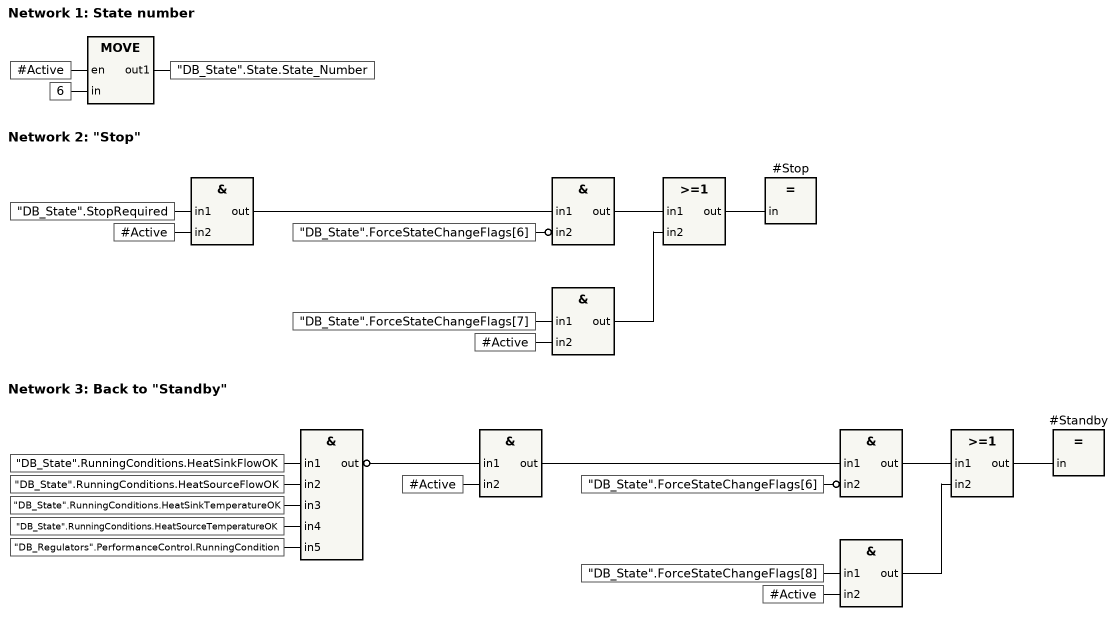
   IF #Active THEN "DB_State".State.State_Number := 6; END_IF;
END_REGION

REGION Network 2: "Stop"
   #Stop := ("DB_State".StopRequired AND #Active AND NOT "DB_State".ForceStateChangeFlags[6]) OR ("DB_State".ForceStateChangeFlags[7] AND #Active);
END_REGION

REGION Network 3: Back to "Standby"
   #Standby := (NOT ("DB_State".RunningConditions.HeatSinkFlowOK AND "DB_State".RunningConditions.HeatSourceFlowOK AND "DB_State".RunningConditions.HeatSinkTemperatureOK AND "DB_State".RunningConditions.HeatSourceTemperatureOK AND "DB_Regulators".PerformanceControl.RunningCondition) AND #Active AND NOT "DB_State".ForceStateChangeFlags[6]) OR ("DB_State".ForceStateChangeFlags[8] AND #Active);
END_REGION
END_FUNCTION

FUNCTION "State7_Stop" : Void   // FC57, FBD
{ S7_Optimized_Access := 'TRUE' }
VERSION : 0.1
// stored: AutoNumber true, IsIECCheckEnabled false, SetENOAutomatically false, UDAEnableTagReadback false
   VAR_INPUT
      Active : Bool;
   END_VAR
   VAR_OUTPUT
      Offline : Bool;
   END_VAR
BEGIN

REGION Network 1: State number
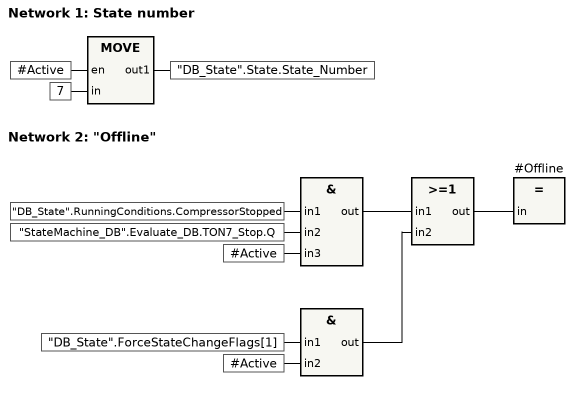
   IF #Active THEN "DB_State".State.State_Number := 7; END_IF;
END_REGION

REGION Network 2: "Offline"
   #Offline := ("DB_State".RunningConditions.CompressorStopped AND "StateMachine_DB".Evaluate_DB.TON7_Stop.Q AND #Active) OR ("DB_State".ForceStateChangeFlags[1] AND #Active);
END_REGION
END_FUNCTION

FUNCTION_BLOCK "ControlAlarmHandling"   // FB19, FBD
{ S7_Optimized_Access := 'TRUE' }
VERSION : 0.1
// stored: AutoNumber true, IsIECCheckEnabled false, IsRetainMemResEnabled false, MemoryReserve 0, SetENOAutomatically false, UDAEnableTagReadback false
   VAR
      A1004 { ExternalAccessible := 'False'; ExternalVisible := 'False'; ExternalWritable := 'False'; S7_SetPoint := 'True'} : "fbHMIEvent";
      A2018 { ExternalAccessible := 'False'; ExternalVisible := 'False'; ExternalWritable := 'False'; S7_SetPoint := 'True'} : "fbHighAlarm";
      A2028 { ExternalAccessible := 'False'; ExternalVisible := 'False'; ExternalWritable := 'False'; S7_SetPoint := 'True'} : "fbLowAlarm";
      A2058 { ExternalAccessible := 'False'; ExternalVisible := 'False'; ExternalWritable := 'False'; S7_SetPoint := 'True'} : "fbLowAlarm";
      A2100 { ExternalAccessible := 'False'; ExternalVisible := 'False'; ExternalWritable := 'False'; S7_SetPoint := 'True'} : "fbHighAlarm";
      A2101 { ExternalAccessible := 'False'; ExternalVisible := 'False'; ExternalWritable := 'False'; S7_SetPoint := 'True'} : "fbHighAlarm";
      A2102 { ExternalAccessible := 'False'; ExternalVisible := 'False'; ExternalWritable := 'False'; S7_SetPoint := 'True'} : "fbHighAlarm";
      A2103 { ExternalAccessible := 'False'; ExternalVisible := 'False'; ExternalWritable := 'False'; S7_SetPoint := 'True'} : "fbHighAlarm";
      A2105 { ExternalAccessible := 'False'; ExternalVisible := 'False'; ExternalWritable := 'False'; S7_SetPoint := 'True'} : "fbHighAlarm";
      A2106 { ExternalAccessible := 'False'; ExternalVisible := 'False'; ExternalWritable := 'False'; S7_SetPoint := 'True'} : "fbHighAlarm";
      A2107 { ExternalAccessible := 'False'; ExternalVisible := 'False'; ExternalWritable := 'False'; S7_SetPoint := 'True'} : "fbHighAlarm";
      A2109 { ExternalAccessible := 'False'; ExternalVisible := 'False'; ExternalWritable := 'False'; S7_SetPoint := 'True'} : "fbHighAlarm";
      A2108 { ExternalAccessible := 'False'; ExternalVisible := 'False'; ExternalWritable := 'False'; S7_SetPoint := 'True'} : "fbHighAlarm";
      A2110 { ExternalAccessible := 'False'; ExternalVisible := 'False'; ExternalWritable := 'False'; S7_SetPoint := 'True'} : "fbHighAlarm";
      A2111 { ExternalAccessible := 'False'; ExternalVisible := 'False'; ExternalWritable := 'False'; S7_SetPoint := 'True'} : "fbHighAlarm";
      A2112 { ExternalAccessible := 'False'; ExternalVisible := 'False'; ExternalWritable := 'False'; S7_SetPoint := 'True'} : "fbHighAlarm";
      A2113 { ExternalAccessible := 'False'; ExternalVisible := 'False'; ExternalWritable := 'False'; S7_SetPoint := 'True'} : "fbHighAlarm";
      A2114 { ExternalAccessible := 'False'; ExternalVisible := 'False'; ExternalWritable := 'False'; S7_SetPoint := 'True'} : "fbHighAlarm";
      A2115 { ExternalAccessible := 'False'; ExternalVisible := 'False'; ExternalWritable := 'False'; S7_SetPoint := 'True'} : "fbLowAlarm";
      A2116 { ExternalAccessible := 'False'; ExternalVisible := 'False'; ExternalWritable := 'False'; S7_SetPoint := 'True'} : "fbHighAlarm";
      A2117 { ExternalAccessible := 'False'; ExternalVisible := 'False'; ExternalWritable := 'False'; S7_SetPoint := 'True'} : "fbLowAlarm";
      A2301 { ExternalAccessible := 'False'; ExternalVisible := 'False'; ExternalWritable := 'False'; S7_SetPoint := 'True'} : "fbLowAlarm";
      A2302 { ExternalAccessible := 'False'; ExternalVisible := 'False'; ExternalWritable := 'False'; S7_SetPoint := 'True'} : "fbHighAlarm";
      A2303 { ExternalAccessible := 'False'; ExternalVisible := 'False'; ExternalWritable := 'False'; S7_SetPoint := 'True'} : "fbHighAlarm";
      A2304 { ExternalAccessible := 'False'; ExternalVisible := 'False'; ExternalWritable := 'False'; S7_SetPoint := 'True'} : "fbLowAlarm";
      A2305 { ExternalAccessible := 'False'; ExternalVisible := 'False'; ExternalWritable := 'False'; S7_SetPoint := 'True'} : "fbHighAlarm";
      A2306 { ExternalAccessible := 'False'; ExternalVisible := 'False'; ExternalWritable := 'False'; S7_SetPoint := 'True'} : "fbHighAlarm";
      A2307 { ExternalAccessible := 'False'; ExternalVisible := 'False'; ExternalWritable := 'False'; S7_SetPoint := 'True'} : "fbHMIEvent";
      A2308 { ExternalAccessible := 'False'; ExternalVisible := 'False'; ExternalWritable := 'False'; S7_SetPoint := 'True'} : "fbHighAlarm";
      A3400 { ExternalAccessible := 'False'; ExternalVisible := 'False'; ExternalWritable := 'False'; S7_SetPoint := 'True'} : "fbHMIEvent";
      A9023 { ExternalAccessible := 'False'; ExternalVisible := 'False'; ExternalWritable := 'False'; S7_SetPoint := 'True'} : "fbDeviationAlarm";
      A9024 { S7_SetPoint := 'True'} : "fbDeviationAlarm";
      A9025 { S7_SetPoint := 'True'} : "fbDeviationAlarm";
      A9026 { S7_SetPoint := 'True'} : "fbDeviationAlarm";
      A9027 { S7_SetPoint := 'True'} : "fbDeviationAlarm";
      A9028 { S7_SetPoint := 'True'} : "fbDeviationAlarm";
      A9029 { S7_SetPoint := 'True'} : "fbDeviationAlarm";
      A9030 { S7_SetPoint := 'True'} : "fbDeviationAlarm";
      A9031 { S7_SetPoint := 'True'} : "fbDeviationAlarm";
   END_VAR
   VAR_TEMP   // added for the SCL form of the ladder/FBD networks
      _w1 : Bool;
   END_VAR
BEGIN

REGION Network 1: 1004
   // DISABLED when no connection
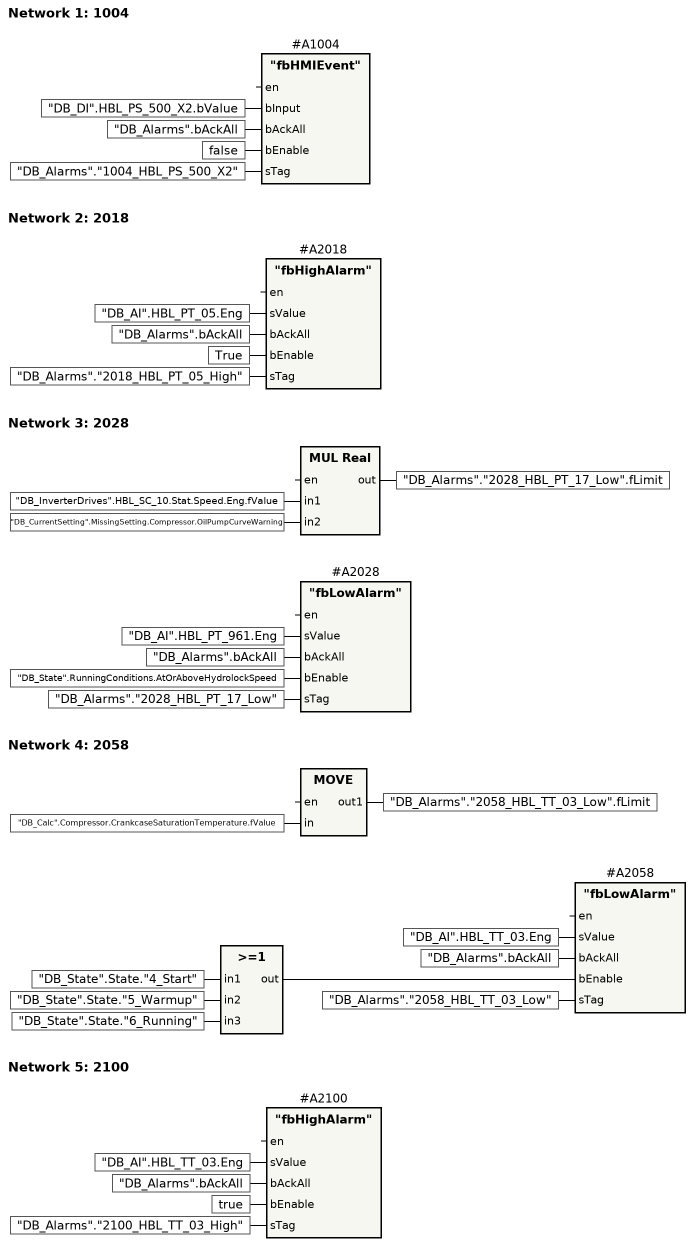
   #A1004(bInput := "DB_DI".HBL_PS_500_X2.bValue,   // "fbHMIEvent"
          bAckAll := "DB_Alarms".bAckAll,
          bEnable := false,
          sTag := "DB_Alarms"."1004_HBL_PS_500_X2");
END_REGION

REGION Network 2: 2018
   #A2018(sValue := "DB_AI".HBL_PT_05.Eng,   // "fbHighAlarm"
          bAckAll := "DB_Alarms".bAckAll,
          bEnable := True,
          sTag := "DB_Alarms"."2018_HBL_PT_05_High");
END_REGION

REGION Network 3: 2028
   // NOTE: alarm limit is dynamic, so don't move it to InitCurrentSettings
   "DB_Alarms"."2028_HBL_PT_17_Low".fLimit := "DB_InverterDrives".HBL_SC_10.Stat.Speed.Eng.fValue * "DB_CurrentSetting".MissingSetting.Compressor.OilPumpCurveWarning;
   #A2028(sValue := "DB_AI".HBL_PT_961.Eng,   // "fbLowAlarm"
          bAckAll := "DB_Alarms".bAckAll,
          bEnable := "DB_State".RunningConditions.AtOrAboveHydrolockSpeed,
          sTag := "DB_Alarms"."2028_HBL_PT_17_Low");
END_REGION

REGION Network 4: 2058
   // NOTE: alarm Low limit is dynamic, so don't move it to InitCurrentSettings
   "DB_Alarms"."2058_HBL_TT_03_Low".fLimit := "DB_Calc".Compressor.CrankcaseSaturationTemperature.fValue;
   #A2058(sValue := "DB_AI".HBL_TT_03.Eng,   // "fbLowAlarm"
          bAckAll := "DB_Alarms".bAckAll,
          bEnable := "DB_State".State."4_Start" OR "DB_State".State."5_Warmup" OR "DB_State".State."6_Running",
          sTag := "DB_Alarms"."2058_HBL_TT_03_Low");
END_REGION

REGION Network 5: 2100
   #A2100(sValue := "DB_AI".HBL_TT_03.Eng,   // "fbHighAlarm"
          bAckAll := "DB_Alarms".bAckAll,
          bEnable := true,
          sTag := "DB_Alarms"."2100_HBL_TT_03_High");
END_REGION

REGION Network 6: 2101
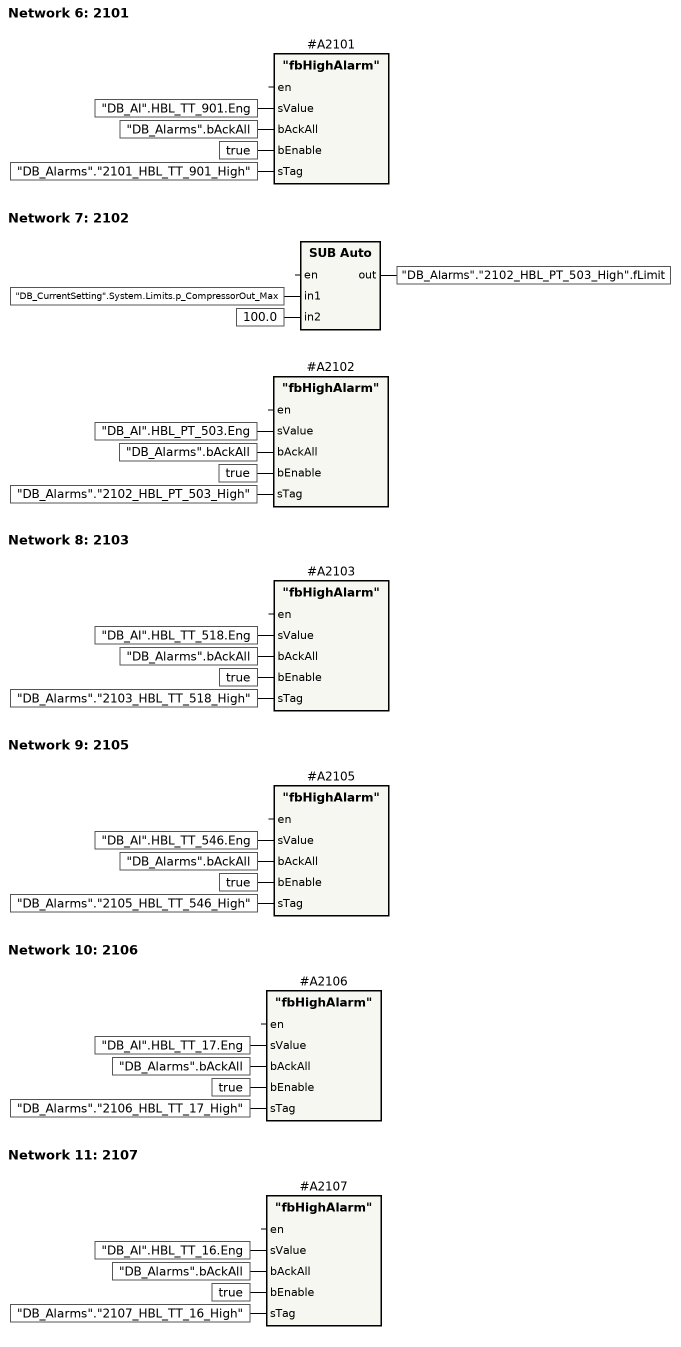
   #A2101(sValue := "DB_AI".HBL_TT_901.Eng,   // "fbHighAlarm"
          bAckAll := "DB_Alarms".bAckAll,
          bEnable := true,
          sTag := "DB_Alarms"."2101_HBL_TT_901_High");
END_REGION

REGION Network 7: 2102
   // Update the alarm limit ALL THE TIME, not just at PLC startup. If the p_CompressorOut_Max value is changed, then this alarms should ALWAYS follow
   "DB_Alarms"."2102_HBL_PT_503_High".fLimit := "DB_CurrentSetting".System.Limits.p_CompressorOut_Max - 100.0;
   #A2102(sValue := "DB_AI".HBL_PT_503.Eng,   // "fbHighAlarm"
          bAckAll := "DB_Alarms".bAckAll,
          bEnable := true,
          sTag := "DB_Alarms"."2102_HBL_PT_503_High");
END_REGION

REGION Network 8: 2103
   #A2103(sValue := "DB_AI".HBL_TT_518.Eng,   // "fbHighAlarm"
          bAckAll := "DB_Alarms".bAckAll,
          bEnable := true,
          sTag := "DB_Alarms"."2103_HBL_TT_518_High");
END_REGION

REGION Network 9: 2105
   #A2105(sValue := "DB_AI".HBL_TT_546.Eng,   // "fbHighAlarm"
          bAckAll := "DB_Alarms".bAckAll,
          bEnable := true,
          sTag := "DB_Alarms"."2105_HBL_TT_546_High");
END_REGION

REGION Network 10: 2106
   #A2106(sValue := "DB_AI".HBL_TT_17.Eng,   // "fbHighAlarm"
          bAckAll := "DB_Alarms".bAckAll,
          bEnable := true,
          sTag := "DB_Alarms"."2106_HBL_TT_17_High");
END_REGION

REGION Network 11: 2107
   #A2107(sValue := "DB_AI".HBL_TT_16.Eng,   // "fbHighAlarm"
          bAckAll := "DB_Alarms".bAckAll,
          bEnable := true,
          sTag := "DB_Alarms"."2107_HBL_TT_16_High");
END_REGION

REGION Network 12: 2108
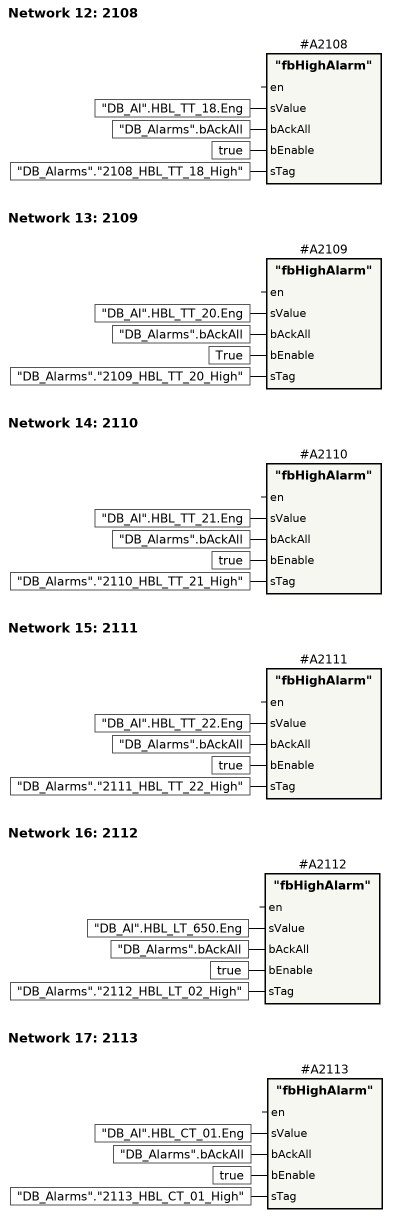
   #A2108(sValue := "DB_AI".HBL_TT_18.Eng,   // "fbHighAlarm"
          bAckAll := "DB_Alarms".bAckAll,
          bEnable := true,
          sTag := "DB_Alarms"."2108_HBL_TT_18_High");
END_REGION

REGION Network 13: 2109
   #A2109(sValue := "DB_AI".HBL_TT_20.Eng,   // "fbHighAlarm"
          bAckAll := "DB_Alarms".bAckAll,
          bEnable := True,
          sTag := "DB_Alarms"."2109_HBL_TT_20_High");
END_REGION

REGION Network 14: 2110
   #A2110(sValue := "DB_AI".HBL_TT_21.Eng,   // "fbHighAlarm"
          bAckAll := "DB_Alarms".bAckAll,
          bEnable := true,
          sTag := "DB_Alarms"."2110_HBL_TT_21_High");
END_REGION

REGION Network 15: 2111
   #A2111(sValue := "DB_AI".HBL_TT_22.Eng,   // "fbHighAlarm"
          bAckAll := "DB_Alarms".bAckAll,
          bEnable := true,
          sTag := "DB_Alarms"."2111_HBL_TT_22_High");
END_REGION

REGION Network 16: 2112
   #A2112(sValue := "DB_AI".HBL_LT_650.Eng,   // "fbHighAlarm"
          bAckAll := "DB_Alarms".bAckAll,
          bEnable := true,
          sTag := "DB_Alarms"."2112_HBL_LT_02_High");
END_REGION

REGION Network 17: 2113
   #A2113(sValue := "DB_AI".HBL_CT_01.Eng,   // "fbHighAlarm"
          bAckAll := "DB_Alarms".bAckAll,
          bEnable := true,
          sTag := "DB_Alarms"."2113_HBL_CT_01_High");
END_REGION

REGION Network 18: 2114
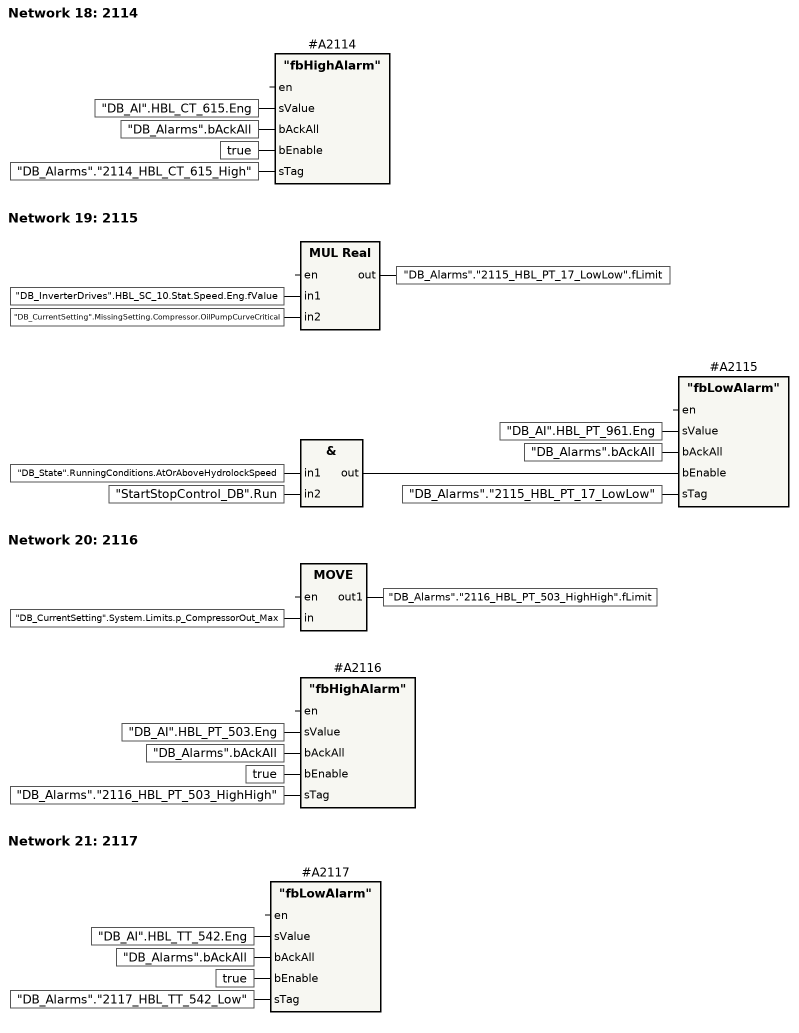
   #A2114(sValue := "DB_AI".HBL_CT_615.Eng,   // "fbHighAlarm"
          bAckAll := "DB_Alarms".bAckAll,
          bEnable := true,
          sTag := "DB_Alarms"."2114_HBL_CT_615_High");
END_REGION

REGION Network 19: 2115
   // NOTE: alarm limit is dynamic, so don't move it to InitCurrentSettings
   "DB_Alarms"."2115_HBL_PT_17_LowLow".fLimit := "DB_InverterDrives".HBL_SC_10.Stat.Speed.Eng.fValue * "DB_CurrentSetting".MissingSetting.Compressor.OilPumpCurveCritical;
   #A2115(sValue := "DB_AI".HBL_PT_961.Eng,   // "fbLowAlarm"
          bAckAll := "DB_Alarms".bAckAll,
          bEnable := "DB_State".RunningConditions.AtOrAboveHydrolockSpeed AND "StartStopControl_DB".Run,
          sTag := "DB_Alarms"."2115_HBL_PT_17_LowLow");
END_REGION

REGION Network 20: 2116
   // Update the alarm limit ALL THE TIME, not just at PLC startup. If the p_CompressorOut_Max value is changed, then this alarms should ALWAYS follow
   "DB_Alarms"."2116_HBL_PT_503_HighHigh".fLimit := "DB_CurrentSetting".System.Limits.p_CompressorOut_Max;
   #A2116(sValue := "DB_AI".HBL_PT_503.Eng,   // "fbHighAlarm"
          bAckAll := "DB_Alarms".bAckAll,
          bEnable := true,
          sTag := "DB_Alarms"."2116_HBL_PT_503_HighHigh");
END_REGION

REGION Network 21: 2117
   #A2117(sValue := "DB_AI".HBL_TT_542.Eng,   // "fbLowAlarm"
          bAckAll := "DB_Alarms".bAckAll,
          bEnable := true,
          sTag := "DB_Alarms"."2117_HBL_TT_542_Low");
END_REGION

REGION Network 22: 2301 & 2302
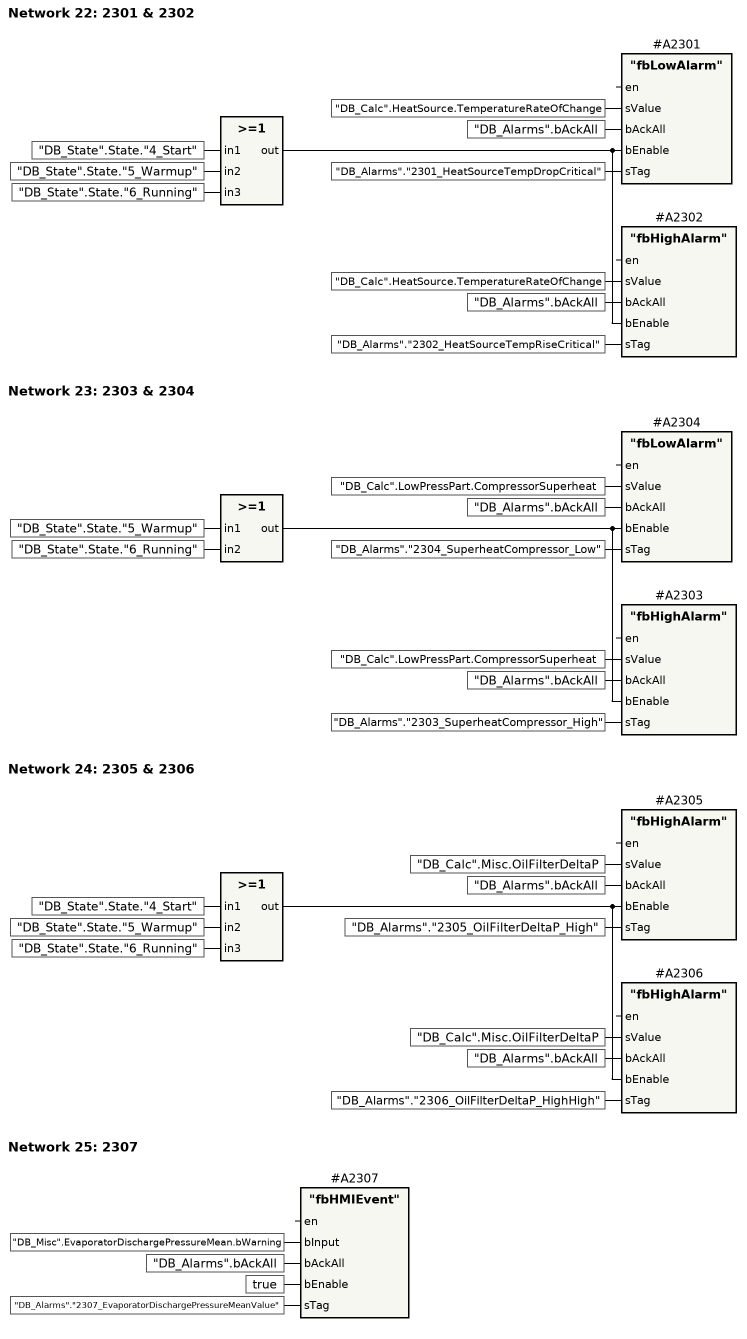
   #_w1 := "DB_State".State."4_Start" OR "DB_State".State."5_Warmup" OR "DB_State".State."6_Running";
   #A2301(sValue := "DB_Calc".HeatSource.TemperatureRateOfChange,   // "fbLowAlarm"
          bAckAll := "DB_Alarms".bAckAll,
          bEnable := #_w1,
          sTag := "DB_Alarms"."2301_HeatSourceTempDropCritical");
   #A2302(sValue := "DB_Calc".HeatSource.TemperatureRateOfChange,   // "fbHighAlarm"
          bAckAll := "DB_Alarms".bAckAll,
          bEnable := #_w1,
          sTag := "DB_Alarms"."2302_HeatSourceTempRiseCritical");
END_REGION

REGION Network 23: 2303 & 2304
   #_w1 := "DB_State".State."5_Warmup" OR "DB_State".State."6_Running";
   #A2304(sValue := "DB_Calc".LowPressPart.CompressorSuperheat,   // "fbLowAlarm"
          bAckAll := "DB_Alarms".bAckAll,
          bEnable := #_w1,
          sTag := "DB_Alarms"."2304_SuperheatCompressor_Low");
   #A2303(sValue := "DB_Calc".LowPressPart.CompressorSuperheat,   // "fbHighAlarm"
          bAckAll := "DB_Alarms".bAckAll,
          bEnable := #_w1,
          sTag := "DB_Alarms"."2303_SuperheatCompressor_High");
END_REGION

REGION Network 24: 2305 & 2306
   #_w1 := "DB_State".State."4_Start" OR "DB_State".State."5_Warmup" OR "DB_State".State."6_Running";
   #A2305(sValue := "DB_Calc".Misc.OilFilterDeltaP,   // "fbHighAlarm"
          bAckAll := "DB_Alarms".bAckAll,
          bEnable := #_w1,
          sTag := "DB_Alarms"."2305_OilFilterDeltaP_High");
   #A2306(sValue := "DB_Calc".Misc.OilFilterDeltaP,   // "fbHighAlarm"
          bAckAll := "DB_Alarms".bAckAll,
          bEnable := #_w1,
          sTag := "DB_Alarms"."2306_OilFilterDeltaP_HighHigh");
END_REGION

REGION Network 25: 2307
   #A2307(bInput := "DB_Misc".EvaporatorDischargePressureMean.bWarning,   // "fbHMIEvent"
          bAckAll := "DB_Alarms".bAckAll,
          bEnable := true,
          sTag := "DB_Alarms"."2307_EvaporatorDischargePressureMeanValue");
END_REGION

REGION Network 26: 2308
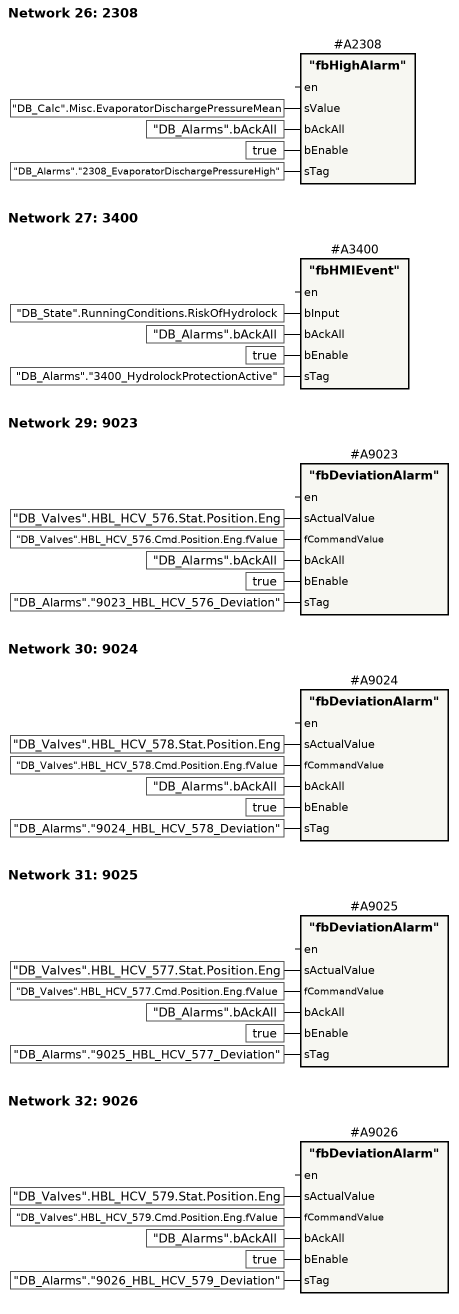
   #A2308(sValue := "DB_Calc".Misc.EvaporatorDischargePressureMean,   // "fbHighAlarm"
          bAckAll := "DB_Alarms".bAckAll,
          bEnable := true,
          sTag := "DB_Alarms"."2308_EvaporatorDischargePressureHigh");
END_REGION

REGION Network 27: 3400
   #A3400(bInput := "DB_State".RunningConditions.RiskOfHydrolock,   // "fbHMIEvent"
          bAckAll := "DB_Alarms".bAckAll,
          bEnable := true,
          sTag := "DB_Alarms"."3400_HydrolockProtectionActive");
END_REGION

REGION Network 28 (SCL): 9023 old
   // This is a deviation alarm, for which a dedicated type does not exist. So we make one here for now with hardocded limits.
   (*
   #A9023(bAckAll := "DB_Alarms".bAckAll, 
           bInput := (ABS(IN := "DB_Valves".HBL_HCV_576.Stat.Position.Eng.fValue -"DB_Valves".HBL_HCV_576.Cmd.Position.Eng.fValue) > 4) OR 
                     ("DB_Valves".HBL_HCV_576.Cmd.Position.Eng.fValue <= 0 AND "DB_Valves".HBL_HCV_576.Stat.Position.Eng.fValue <2),
           sTag := "DB_Alarms"."9023_ExpansionValveDeviation");

   *)
END_REGION

REGION Network 29: 9023
   #A9023(sActualValue := "DB_Valves".HBL_HCV_576.Stat.Position.Eng,   // "fbDeviationAlarm"
          fCommandValue := "DB_Valves".HBL_HCV_576.Cmd.Position.Eng.fValue,
          bAckAll := "DB_Alarms".bAckAll,
          bEnable := true,
          sTag := "DB_Alarms"."9023_HBL_HCV_576_Deviation");
END_REGION

REGION Network 30: 9024
   #A9024(sActualValue := "DB_Valves".HBL_HCV_578.Stat.Position.Eng,   // "fbDeviationAlarm"
          fCommandValue := "DB_Valves".HBL_HCV_578.Cmd.Position.Eng.fValue,
          bAckAll := "DB_Alarms".bAckAll,
          bEnable := true,
          sTag := "DB_Alarms"."9024_HBL_HCV_578_Deviation");
END_REGION

REGION Network 31: 9025
   #A9025(sActualValue := "DB_Valves".HBL_HCV_577.Stat.Position.Eng,   // "fbDeviationAlarm"
          fCommandValue := "DB_Valves".HBL_HCV_577.Cmd.Position.Eng.fValue,
          bAckAll := "DB_Alarms".bAckAll,
          bEnable := true,
          sTag := "DB_Alarms"."9025_HBL_HCV_577_Deviation");
END_REGION

REGION Network 32: 9026
   #A9026(sActualValue := "DB_Valves".HBL_HCV_579.Stat.Position.Eng,   // "fbDeviationAlarm"
          fCommandValue := "DB_Valves".HBL_HCV_579.Cmd.Position.Eng.fValue,
          bAckAll := "DB_Alarms".bAckAll,
          bEnable := true,
          sTag := "DB_Alarms"."9026_HBL_HCV_579_Deviation");
END_REGION

REGION Network 33: 9027
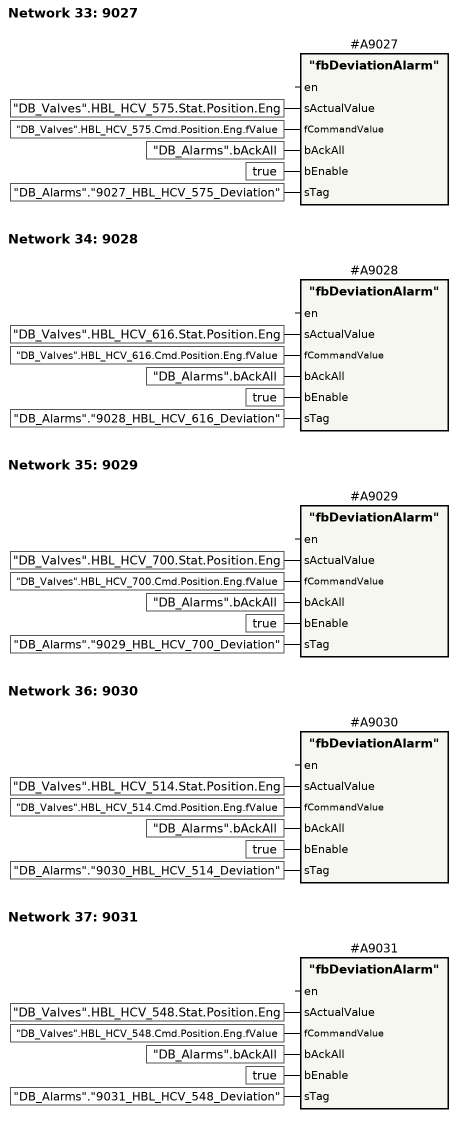
   #A9027(sActualValue := "DB_Valves".HBL_HCV_575.Stat.Position.Eng,   // "fbDeviationAlarm"
          fCommandValue := "DB_Valves".HBL_HCV_575.Cmd.Position.Eng.fValue,
          bAckAll := "DB_Alarms".bAckAll,
          bEnable := true,
          sTag := "DB_Alarms"."9027_HBL_HCV_575_Deviation");
END_REGION

REGION Network 34: 9028
   #A9028(sActualValue := "DB_Valves".HBL_HCV_616.Stat.Position.Eng,   // "fbDeviationAlarm"
          fCommandValue := "DB_Valves".HBL_HCV_616.Cmd.Position.Eng.fValue,
          bAckAll := "DB_Alarms".bAckAll,
          bEnable := true,
          sTag := "DB_Alarms"."9028_HBL_HCV_616_Deviation");
END_REGION

REGION Network 35: 9029
   #A9029(sActualValue := "DB_Valves".HBL_HCV_700.Stat.Position.Eng,   // "fbDeviationAlarm"
          fCommandValue := "DB_Valves".HBL_HCV_700.Cmd.Position.Eng.fValue,
          bAckAll := "DB_Alarms".bAckAll,
          bEnable := true,
          sTag := "DB_Alarms"."9029_HBL_HCV_700_Deviation");
END_REGION

REGION Network 36: 9030
   #A9030(sActualValue := "DB_Valves".HBL_HCV_514.Stat.Position.Eng,   // "fbDeviationAlarm"
          fCommandValue := "DB_Valves".HBL_HCV_514.Cmd.Position.Eng.fValue,
          bAckAll := "DB_Alarms".bAckAll,
          bEnable := true,
          sTag := "DB_Alarms"."9030_HBL_HCV_514_Deviation");
END_REGION

REGION Network 37: 9031
   #A9031(sActualValue := "DB_Valves".HBL_HCV_548.Stat.Position.Eng,   // "fbDeviationAlarm"
          fCommandValue := "DB_Valves".HBL_HCV_548.Cmd.Position.Eng.fValue,
          bAckAll := "DB_Alarms".bAckAll,
          bEnable := true,
          sTag := "DB_Alarms"."9031_HBL_HCV_548_Deviation");
END_REGION
END_FUNCTION_BLOCK

FUNCTION_BLOCK "fbHighAlarm"   // FB31, FBD
TITLE = Lightweight version of fbAnalogAlarm with only one limit
{ S7_Optimized_Access := 'TRUE' }
VERSION : 0.1
// stored: AutoNumber true, IsIECCheckEnabled false, IsRetainMemResEnabled false, MemoryReserve 0, SetENOAutomatically false, UDAEnableTagReadback false
   VAR_INPUT
      sValue : "stCalcValue";
      bAckAll : Bool;
      bEnable : Bool;
   END_VAR
   VAR_IN_OUT
      sTag : "stLimitAlarm";
   END_VAR
   VAR
      Alarm : "fbLimitAlarm";
   END_VAR
   VAR CONSTANT
      Low : Bool;
      High : Bool := true;
   END_VAR
BEGIN

REGION Network 1
   // Note that alarm is disabled if CalcValue .bError is set
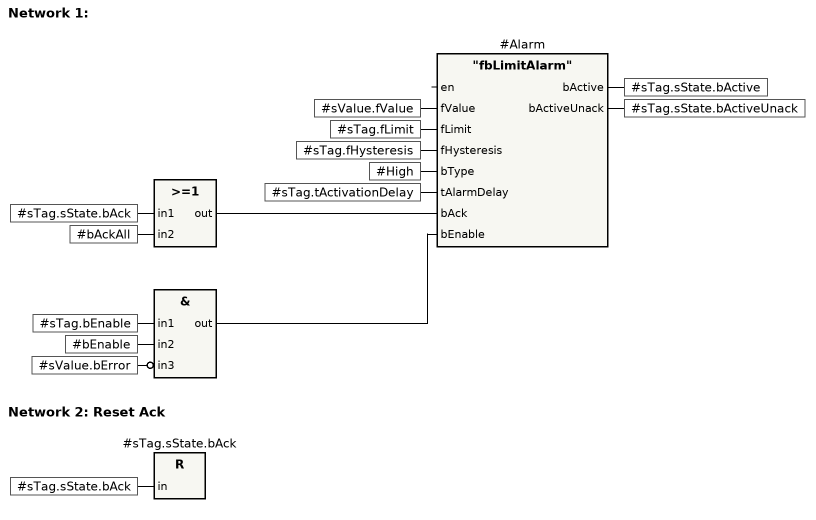
   #Alarm(fValue := #sValue.fValue,   // "fbLimitAlarm"
          fLimit := #sTag.fLimit,
          fHysteresis := #sTag.fHysteresis,
          bType := #High,
          tAlarmDelay := #sTag.tActivationDelay,
          bAck := #sTag.sState.bAck OR #bAckAll,
          bEnable := #sTag.bEnable AND #bEnable AND NOT #sValue.bError,
          bActive => #sTag.sState.bActive,
          bActiveUnack => #sTag.sState.bActiveUnack);
END_REGION

REGION Network 2: Reset Ack
   IF #sTag.sState.bAck THEN #sTag.sState.bAck := FALSE; END_IF;
END_REGION
END_FUNCTION_BLOCK

FUNCTION_BLOCK "fbLimitAlarm"   // FB46, FBD
{ S7_Optimized_Access := 'TRUE' }
VERSION : 0.1
// stored: AutoNumber true, IsIECCheckEnabled false, IsRetainMemResEnabled false, MemoryReserve 0, SetENOAutomatically false, UDAEnableTagReadback false
   VAR_INPUT
      fValue : Real;
      fLimit : Real;
      fHysteresis : Real;
      bType : Bool;
      tAlarmDelay : Time;
      bAck : Bool;
      bEnable : Bool;
   END_VAR
   VAR_OUTPUT
      bActive : Bool;
      bActiveUnack : Bool;
   END_VAR
   VAR
      Limit : "fbHysteresis";
      Alarm { S7_SetPoint := 'True'} : "fbAlarm";
   END_VAR
   VAR_TEMP
      AlarmCondition : Bool;
   END_VAR
BEGIN

REGION Network 1: Check for alarm condition
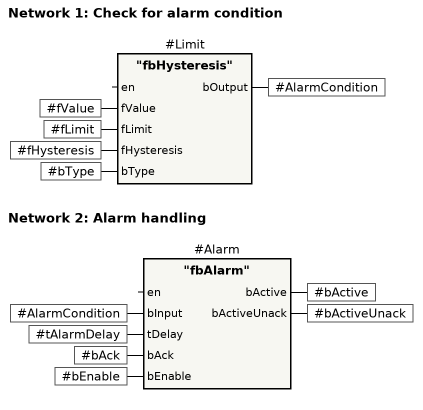
   #Limit(fValue := #fValue,   // "fbHysteresis"
          fLimit := #fLimit,
          fHysteresis := #fHysteresis,
          bType := #bType,
          bOutput => #AlarmCondition);
END_REGION

REGION Network 2: Alarm handling
   #Alarm(bInput := #AlarmCondition,   // "fbAlarm"
          tDelay := #tAlarmDelay,
          bAck := #bAck,
          bEnable := #bEnable,
          bActive => #bActive,
          bActiveUnack => #bActiveUnack);
END_REGION
END_FUNCTION_BLOCK

FUNCTION_BLOCK "fbHysteresis"   // FB43, FBD
TITLE = Threshold detection with deadband
{ S7_Optimized_Access := 'TRUE' }
VERSION : 0.1
// stored: AutoNumber true, IsIECCheckEnabled false, IsRetainMemResEnabled false, MemoryReserve 0, SetENOAutomatically false, UDAEnableTagReadback false
   VAR_INPUT
      fValue : Real;
      fLimit : Real;
      fHysteresis : Real;
      bType : Bool;   // 0 = under the limit, 1 = over the limit
   END_VAR
   VAR_OUTPUT
      bOutput : Bool;
   END_VAR
   VAR
      State : Bool;
   END_VAR
   VAR_TEMP
      Set : Bool;
      Reset : Bool;
   END_VAR
BEGIN

REGION Network 1 (SCL)
   // Over the limit: 
   //  - output is activated when input value is greater than the limit plus half the deadband, AND STAYS ACTIVATED UNTIL the deactivation condition is reached
   //  - output is deactivated when the input value is less than the limit minus half the deadband, AND STAYS DEACTIVATED UNTIL the activation condition is reached
   // 
   // Under the limit: 
   //  - output is activated when the input value is less than the limit minus half the deadband
   //  - output is deactivated when the input value is greater than the limit plus half the deadband
   IF #bType = TRUE THEN
       #Set := #fValue > (#fLimit + #fHysteresis/2);
       #Reset := #fValue < (#fLimit - #fHysteresis/2);
   ELSE
       #Set := #fValue < (#fLimit - #fHysteresis/2);
       #Reset := #fValue > (#fLimit + #fHysteresis/2);
   END_IF;
END_REGION

REGION Network 2
   // A memory bit preserves the output state, even when the input changes. You can't have hysteresis without memory!
